//     Drive/Outputs/Out/nCtrl1 @bit 2 <-> STM Control/Control/Reduce torque
//     Drive/Outputs/Out/nCtrl1 @bit 1 <-> STM Control/Control/Reset
//     Drive/Outputs/Out/nDataOut2[0] <-> STM Velocity/Velocity
//   (this object) <-> PLC Rail (EtherCAT)/Power (EK1200)/PLC Junction 2 (EK1122)/IM2L0 AT2L0 SL1L0 JUNCTION (CU1124)/X1 PF1L0-WFS (EK1100)/PF1L0-EL5042
//     Enc/Inputs/In/nComState @bit 1 <-> WcState/InputToggle
//     Enc/Inputs/In/nComState <-> WcState/WcState
//     Enc/Inputs/In/nDataIn1 <-> FB Inputs Channel 2/Position
//     Enc/Inputs/In/nState1 @bit 12 <-> FB Inputs Channel 2/Status/Diag
//     Enc/Inputs/In/nState1 @bit 1 <-> FB Inputs Channel 2/Status/Error
//     Enc/Inputs/In/nState1 @bit 14 <-> FB Inputs Channel 2/Status/Input cycle counter
//     Enc/Inputs/In/nState1 @bit 2 <-> FB Inputs Channel 2/Status/Ready
//     Enc/Inputs/In/nState1 @bit 13 <-> FB Inputs Channel 2/Status/TxPDO State
//     Enc/Inputs/In/nState1 <-> FB Inputs Channel 2/Status/Warning
//   (this object) <-> PLC Rail (EtherCAT)/Power (EK1200)/PLC Junction 2 (EK1122)/IM2L0 AT2L0 SL1L0 JUNCTION (CU1124)/X1 PF1L0-WFS (EK1100)/PF1L0-EL7041-01
//     Drive/Inputs/In/nState1 @bit 3 <-> STM Status/Status/Error
//     Drive/Inputs/In/nState1 @bit 5 <-> STM Status/Status/Moving negative
//     Drive/Inputs/In/nState1 @bit 4 <-> STM Status/Status/Moving positive
//     Drive/Inputs/In/nState1 @bit 1 <-> STM Status/Status/Ready
//     Drive/Inputs/In/nState1 <-> STM Status/Status/Ready to enable
//     Drive/Inputs/In/nState1 @bit 6 <-> STM Status/Status/Torque reduced
//     Drive/Inputs/In/nState1 @bit 2 <-> STM Status/Status/Warning
//     Drive/Inputs/In/nState2 @bit 3 <-> STM Status/Status/Digital input 1
//     Drive/Inputs/In/nState2 @bit 4 <-> STM Status/Status/Digital input 2
//     Drive/Inputs/In/nState2 @bit 5 <-> STM Status/Status/Sync error
//     Drive/Inputs/In/nState2 @bit 7 <-> STM Status/Status/TxPDO Toggle
//     Drive/Inputs/In/nState4 @bit 1 <-> WcState/InputToggle
//     Drive/Inputs/In/nState4 <-> WcState/WcState
//     Drive/Outputs/Out/nCtrl1 <-> STM Control/Control/Enable
//     Drive/Outputs/Out/nCtrl1 @bit 2 <-> STM Control/Control/Reduce torque
//     Drive/Outputs/Out/nCtrl1 @bit 1 <-> STM Control/Control/Reset
//     Drive/Outputs/Out/nDataOut2[0] <-> STM Velocity/Velocity
//   (this object) <-> PLC Rail (EtherCAT)/Power (EK1200)/PLC Junction 1 (EK1122)/X1 RTDSL0 (EK1100)/RTDSL0-EL7041-01
//     Drive/Inputs/In/nState1 @bit 3 <-> STM Status/Status/Error
//     Drive/Inputs/In/nState1 @bit 5 <-> STM Status/Status/Moving negative
//     Drive/Inputs/In/nState1 @bit 4 <-> STM Status/Status/Moving positive
//     Drive/Inputs/In/nState1 @bit 1 <-> STM Status/Status/Ready
//     Drive/Inputs/In/nState1 <-> STM Status/Status/Ready to enable
//     Drive/Inputs/In/nState1 @bit 6 <-> STM Status/Status/Torque reduced
//     Drive/Inputs/In/nState1 @bit 2 <-> STM Status/Status/Warning
//     Drive/Inputs/In/nState2 @bit 3 <-> STM Status/Status/Digital input 1
//     Drive/Inputs/In/nState2 @bit 4 <-> STM Status/Status/Digital input 2
//     Drive/Inputs/In/nState2 @bit 5 <-> STM Status/Status/Sync error
//     Drive/Inputs/In/nState2 @bit 7 <-> STM Status/Status/TxPDO Toggle
//     Drive/Inputs/In/nState4 @bit 1 <-> WcState/InputToggle
//     Drive/Inputs/In/nState4 <-> WcState/WcState
//     Drive/Outputs/Out/nCtrl1 <-> STM Control/Control/Enable
//     Drive/Outputs/Out/nCtrl1 @bit 2 <-> STM Control/Control/Reduce torque
//     Drive/Outputs/Out/nCtrl1 @bit 1 <-> STM Control/Control/Reset
//     Drive/Outputs/Out/nDataOut2[0] <-> STM Velocity/Velocity
//     Enc/Inputs/In/nDataIn1[0] <-> ENC Status compact/Counter value
//     Enc/Inputs/In/nDataIn2[0] <-> ENC Status compact/Latch value
//     Enc/Inputs/In/nState1 @bit 4 <-> ENC Status compact/Status/Counter overflow
//     Enc/Inputs/In/nState1 @bit 3 <-> ENC Status compact/Status/Counter underflow
//     Enc/Inputs/In/nState1 @bit 7 <-> ENC Status compact/Status/Extrapolation stall
//     Enc/Inputs/In/nState1 <-> ENC Status compact/Status/Latch C valid
//     Enc/Inputs/In/nState1 @bit 1 <-> ENC Status compact/Status/Latch extern valid
//     Enc/Inputs/In/nState1 @bit 2 <-> ENC Status compact/Status/Set counter done
//     Enc/Inputs/In/nState2 @bit 4 <-> ENC Status compact/Status/Status of extern latch
//     Enc/Inputs/In/nState2 <-> ENC Status compact/Status/Status of input A
//     Enc/Inputs/In/nState2 @bit 1 <-> ENC Status compact/Status/Status of input B
//     Enc/Inputs/In/nState2 @bit 2 <-> ENC Status compact/Status/Status of input C
//     Enc/Inputs/In/nState2 @bit 5 <-> ENC Status compact/Status/Sync error
//     Enc/Inputs/In/nState2 @bit 7 <-> ENC Status compact/Status/TxPDO Toggle
//     Enc/Inputs/In/nState4 @bit 1 <-> WcState/InputToggle
//     Enc/Inputs/In/nState4 <-> WcState/WcState
//     Enc/Outputs/Out/nCtrl1 <-> ENC Control compact/Control/Enable latch C
//     Enc/Outputs/Out/nCtrl1 @bit 3 <-> ENC Control compact/Control/Enable latch extern on negative edge
//     Enc/Outputs/Out/nCtrl1 @bit 1 <-> ENC Control compact/Control/Enable latch extern on positive edge
//     Enc/Outputs/Out/nCtrl1 @bit 2 <-> ENC Control compact/Control/Set counter
//     Enc/Outputs/Out/nDataOut1[0] <-> ENC Control compact/Set counter value
//   (this object) <-> PLC Rail (EtherCAT)/Power (EK1200)/PLC Junction 1 (EK1122)/X1 RTDSL0 (EK1100)/RTDSL0-EL7041-05
//     Drive/Inputs/In/nState1 @bit 3 <-> STM Status/Status/Error
//     Drive/Inputs/In/nState1 @bit 5 <-> STM Status/Status/Moving negative
//     Drive/Inputs/In/nState1 @bit 4 <-> STM Status/Status/Moving positive
//     Drive/Inputs/In/nState1 @bit 1 <-> STM Status/Status/Ready
//     Drive/Inputs/In/nState1 <-> STM Status/Status/Ready to enable
//     Drive/Inputs/In/nState1 @bit 6 <-> STM Status/Status/Torque reduced
//     Drive/Inputs/In/nState1 @bit 2 <-> STM Status/Status/Warning
//     Drive/Inputs/In/nState2 @bit 3 <-> STM Status/Status/Digital input 1
//     Drive/Inputs/In/nState2 @bit 4 <-> STM Status/Status/Digital input 2
//     Drive/Inputs/In/nState2 @bit 5 <-> STM Status/Status/Sync error
//     Drive/Inputs/In/nState2 @bit 7 <-> STM Status/Status/TxPDO Toggle
//     Drive/Inputs/In/nState4 @bit 1 <-> WcState/InputToggle
//     Drive/Inputs/In/nState4 <-> WcState/WcState
//     Drive/Outputs/Out/nCtrl1 <-> STM Control/Control/Enable
//     Drive/Outputs/Out/nCtrl1 @bit 2 <-> STM Control/Control/Reduce torque
//     Drive/Outputs/Out/nCtrl1 @bit 1 <-> STM Control/Control/Reset
//     Drive/Outputs/Out/nDataOut2[0] <-> STM Velocity/Velocity
//   (this object) <-> PLC Rail (EtherCAT)/Power (EK1200)/PLC Junction 1 (EK1122)/X1 RTDSL0 (EK1100)/Term 113 (EL3054)
//     Enc/Inputs/In/nDataIn1[0] <-> AI Standard Channel 1/Value
//     Enc/Inputs/In/nState4 @bit 1 <-> WcState/InputToggle
//     Enc/Inputs/In/nState4 <-> WcState/WcState
//   (this object) <-> PLC Rail (EtherCAT)/Power (EK1200)/PLC Junction 2 (EK1122)/IM2L0 AT2L0 SL1L0 JUNCTION (CU1124)/X1 SL1L0-Power (EK1100)/SL1L0-EL5042-E2
//     Enc/Inputs/In/nComState @bit 1 <-> WcState/InputToggle
//     Enc/Inputs/In/nComState <-> WcState/WcState
//     Enc/Inputs/In/nDataIn1 <-> FB Inputs Channel 1/Position
//     Enc/Inputs/In/nDataIn1 <-> FB Inputs Channel 2/Position
//     Enc/Inputs/In/nState1 @bit 12 <-> FB Inputs Channel 1/Status/Diag
//     Enc/Inputs/In/nState1 @bit 12 <-> FB Inputs Channel 2/Status/Diag
//     Enc/Inputs/In/nState1 @bit 1 <-> FB Inputs Channel 1/Status/Error
//     Enc/Inputs/In/nState1 @bit 1 <-> FB Inputs Channel 2/Status/Error
//     Enc/Inputs/In/nState1 @bit 14 <-> FB Inputs Channel 1/Status/Input cycle counter
//     Enc/Inputs/In/nState1 @bit 14 <-> FB Inputs Channel 2/Status/Input cycle counter
//     Enc/Inputs/In/nState1 @bit 2 <-> FB Inputs Channel 1/Status/Ready
//     Enc/Inputs/In/nState1 @bit 2 <-> FB Inputs Channel 2/Status/Ready
//     Enc/Inputs/In/nState1 @bit 13 <-> FB Inputs Channel 1/Status/TxPDO State
//     Enc/Inputs/In/nState1 @bit 13 <-> FB Inputs Channel 2/Status/TxPDO State
//     Enc/Inputs/In/nState1 <-> FB Inputs Channel 1/Status/Warning
//     Enc/Inputs/In/nState1 <-> FB Inputs Channel 2/Status/Warning
//   (this object) <-> PLC Rail (EtherCAT)/Power (EK1200)/PLC Junction 2 (EK1122)/IM2L0 AT2L0 SL1L0 JUNCTION (CU1124)/X1 SL1L0-Power (EK1100)/SL1L0-EL7041-E1
//     Drive/Inputs/In/nState1 @bit 3 <-> STM Status/Status/Error
//     Drive/Inputs/In/nState1 @bit 5 <-> STM Status/Status/Moving negative
//     Drive/Inputs/In/nState1 @bit 4 <-> STM Status/Status/Moving positive
//     Drive/Inputs/In/nState1 @bit 1 <-> STM Status/Status/Ready
//     Drive/Inputs/In/nState1 <-> STM Status/Status/Ready to enable
//     Drive/Inputs/In/nState1 @bit 6 <-> STM Status/Status/Torque reduced
//     Drive/Inputs/In/nState1 @bit 2 <-> STM Status/Status/Warning
//     Drive/Inputs/In/nState2 @bit 3 <-> STM Status/Status/Digital input 1
//     Drive/Inputs/In/nState2 @bit 4 <-> STM Status/Status/Digital input 2
//     Drive/Inputs/In/nState2 @bit 5 <-> STM Status/Status/Sync error
//     Drive/Inputs/In/nState2 @bit 7 <-> STM Status/Status/TxPDO Toggle
//     Drive/Inputs/In/nState4 @bit 1 <-> WcState/InputToggle
//     Drive/Inputs/In/nState4 <-> WcState/WcState
//     Drive/Outputs/Out/nCtrl1 <-> STM Control/Control/Enable
//     Drive/Outputs/Out/nCtrl1 @bit 2 <-> STM Control/Control/Reduce torque
//     Drive/Outputs/Out/nCtrl1 @bit 1 <-> STM Control/Control/Reset
//     Drive/Outputs/Out/nDataOut2[0] <-> STM Velocity/Velocity
//   (this object) <-> PLC Rail (EtherCAT)/Power (EK1200)/PLC Junction 2 (EK1122)/IM2L0 AT2L0 SL1L0 JUNCTION (CU1124)/X1 SL1L0-Power (EK1100)/SL1L0-EL7041-E3
//     Drive/Inputs/In/nState1 @bit 3 <-> STM Status/Status/Error
//     Drive/Inputs/In/nState1 @bit 5 <-> STM Status/Status/Moving negative
//     Drive/Inputs/In/nState1 @bit 4 <-> STM Status/Status/Moving positive
//     Drive/Inputs/In/nState1 @bit 1 <-> STM Status/Status/Ready
//     Drive/Inputs/In/nState1 <-> STM Status/Status/Ready to enable
//     Drive/Inputs/In/nState1 @bit 6 <-> STM Status/Status/Torque reduced
//     Drive/Inputs/In/nState1 @bit 2 <-> STM Status/Status/Warning
//     Drive/Inputs/In/nState2 @bit 3 <-> STM Status/Status/Digital input 1
//     Drive/Inputs/In/nState2 @bit 4 <-> STM Status/Status/Digital input 2
//     Drive/Inputs/In/nState2 @bit 5 <-> STM Status/Status/Sync error
//     Drive/Inputs/In/nState2 @bit 7 <-> STM Status/Status/TxPDO Toggle
//     Drive/Inputs/In/nState4 @bit 1 <-> WcState/InputToggle
//     Drive/Inputs/In/nState4 <-> WcState/WcState
//     Drive/Outputs/Out/nCtrl1 <-> STM Control/Control/Enable
//     Drive/Outputs/Out/nCtrl1 @bit 2 <-> STM Control/Control/Reduce torque
//     Drive/Outputs/Out/nCtrl1 @bit 1 <-> STM Control/Control/Reset
//     Drive/Outputs/Out/nDataOut2[0] <-> STM Velocity/Velocity
//   (this object) <-> PLC Rail (EtherCAT)/Power (EK1200)/PLC Junction 2 (EK1122)/IM2L0 AT2L0 SL1L0 JUNCTION (CU1124)/X1 SL1L0-Power (EK1100)/SL1L0-EL5042-E6
//     Enc/Inputs/In/nComState @bit 1 <-> WcState/InputToggle
//     Enc/Inputs/In/nComState <-> WcState/WcState
//     Enc/Inputs/In/nDataIn1 <-> FB Inputs Channel 1/Position
//     Enc/Inputs/In/nDataIn1 <-> FB Inputs Channel 2/Position
//     Enc/Inputs/In/nState1 @bit 12 <-> FB Inputs Channel 1/Status/Diag
//     Enc/Inputs/In/nState1 @bit 12 <-> FB Inputs Channel 2/Status/Diag
//     Enc/Inputs/In/nState1 @bit 1 <-> FB Inputs Channel 1/Status/Error
//     Enc/Inputs/In/nState1 @bit 1 <-> FB Inputs Channel 2/Status/Error
//     Enc/Inputs/In/nState1 @bit 14 <-> FB Inputs Channel 1/Status/Input cycle counter
//     Enc/Inputs/In/nState1 @bit 14 <-> FB Inputs Channel 2/Status/Input cycle counter
//     Enc/Inputs/In/nState1 @bit 2 <-> FB Inputs Channel 1/Status/Ready
//     Enc/Inputs/In/nState1 @bit 2 <-> FB Inputs Channel 2/Status/Ready
//     Enc/Inputs/In/nState1 @bit 13 <-> FB Inputs Channel 1/Status/TxPDO State
//     Enc/Inputs/In/nState1 @bit 13 <-> FB Inputs Channel 2/Status/TxPDO State
//     Enc/Inputs/In/nState1 <-> FB Inputs Channel 1/Status/Warning
//     Enc/Inputs/In/nState1 <-> FB Inputs Channel 2/Status/Warning
//   (this object) <-> PLC Rail (EtherCAT)/Power (EK1200)/PLC Junction 2 (EK1122)/IM2L0 AT2L0 SL1L0 JUNCTION (CU1124)/X1 SL1L0-Power (EK1100)/SL1L0-EL7041-E5
//     Drive/Inputs/In/nState1 @bit 3 <-> STM Status/Status/Error
//     Drive/Inputs/In/nState1 @bit 5 <-> STM Status/Status/Moving negative
//     Drive/Inputs/In/nState1 @bit 4 <-> STM Status/Status/Moving positive
//     Drive/Inputs/In/nState1 @bit 1 <-> STM Status/Status/Ready
//     Drive/Inputs/In/nState1 <-> STM Status/Status/Ready to enable
//     Drive/Inputs/In/nState1 @bit 6 <-> STM Status/Status/Torque reduced
//     Drive/Inputs/In/nState1 @bit 2 <-> STM Status/Status/Warning
//     Drive/Inputs/In/nState2 @bit 3 <-> STM Status/Status/Digital input 1
//     Drive/Inputs/In/nState2 @bit 4 <-> STM Status/Status/Digital input 2
//     Drive/Inputs/In/nState2 @bit 5 <-> STM Status/Status/Sync error
//     Drive/Inputs/In/nState2 @bit 7 <-> STM Status/Status/TxPDO Toggle
//     Drive/Inputs/In/nState4 @bit 1 <-> WcState/InputToggle
//     Drive/Inputs/In/nState4 <-> WcState/WcState
//     Drive/Outputs/Out/nCtrl1 <-> STM Control/Control/Enable
//     Drive/Outputs/Out/nCtrl1 @bit 2 <-> STM Control/Control/Reduce torque
//     Drive/Outputs/Out/nCtrl1 @bit 1 <-> STM Control/Control/Reset
//     Drive/Outputs/Out/nDataOut2[0] <-> STM Velocity/Velocity
//   (this object) <-> PLC Rail (EtherCAT)/Power (EK1200)/PLC Junction 2 (EK1122)/IM2L0 AT2L0 SL1L0 JUNCTION (CU1124)/X1 SL1L0-Power (EK1100)/SL1L0-EL7041-E7
//     Drive/Inputs/In/nState1 @bit 3 <-> STM Status/Status/Error
//     Drive/Inputs/In/nState1 @bit 5 <-> STM Status/Status/Moving negative
//     Drive/Inputs/In/nState1 @bit 4 <-> STM Status/Status/Moving positive
//     Drive/Inputs/In/nState1 @bit 1 <-> STM Status/Status/Ready
//     Drive/Inputs/In/nState1 <-> STM Status/Status/Ready to enable
//     Drive/Inputs/In/nState1 @bit 6 <-> STM Status/Status/Torque reduced
//     Drive/Inputs/In/nState1 @bit 2 <-> STM Status/Status/Warning
//     Drive/Inputs/In/nState2 @bit 3 <-> STM Status/Status/Digital input 1
//     Drive/Inputs/In/nState2 @bit 4 <-> STM Status/Status/Digital input 2
//     Drive/Inputs/In/nState2 @bit 5 <-> STM Status/Status/Sync error
//     Drive/Inputs/In/nState2 @bit 7 <-> STM Status/Status/TxPDO Toggle
//     Drive/Inputs/In/nState4 @bit 1 <-> WcState/InputToggle
//     Drive/Inputs/In/nState4 <-> WcState/WcState
//     Drive/Outputs/Out/nCtrl1 <-> STM Control/Control/Enable
//     Drive/Outputs/Out/nCtrl1 @bit 2 <-> STM Control/Control/Reduce torque
//     Drive/Outputs/Out/nCtrl1 @bit 1 <-> STM Control/Control/Reset
//     Drive/Outputs/Out/nDataOut2[0] <-> STM Velocity/Velocity
//   lfe_motion Instance <-> PLC Rail (EtherCAT)/Power (EK1200)/PLC Junction 1 (EK1122)/X1 RTDSL0 (EK1100)/RTDSL0-EL7041-01
//     PlcTask Inputs/Main.M33.bLimitBackwardEnable <-> STM Status/Status/Digital input 2
//     PlcTask Inputs/Main.M33.bLimitForwardEnable <-> STM Status/Status/Digital input 1
//   lfe_motion Instance <-> PLC Rail (EtherCAT)/Power (EK1200)/PLC Junction 1 (EK1122)/X1 RTDSL0 (EK1100)/RTDSL0-EL7041-05
//     PlcTask Inputs/Main.M38.bLimitBackwardEnable <-> STM Status/Status/Digital input 2
//     PlcTask Inputs/Main.M38.bLimitForwardEnable <-> STM Status/Status/Digital input 1
//   lfe_motion Instance <-> PLC Rail (EtherCAT)/Power (EK1200)/PLC Junction 1 (EK1122)/X1 RTDSL0 (EK1100)/RTDSL0-MPA-EL1008
//     PlcTask Inputs/RTDSL0.RTDSL0_MPA_01.i_xInsertedLS <-> Channel 1/Input
//     PlcTask Inputs/RTDSL0.RTDSL0_MPA_02.i_xInsertedLS <-> Channel 3/Input
//     PlcTask Inputs/RTDSL0.RTDSL0_MPA_03.i_xInsertedLS <-> Channel 5/Input
//     PlcTask Inputs/RTDSL0.RTDSL0_MPA_04.i_xInsertedLS <-> Channel 7/Input
//     PlcTask Inputs/RTDSL0.RTDSL0_MPA_01.i_xRetractedLS <-> Channel 2/Input
//     PlcTask Inputs/RTDSL0.RTDSL0_MPA_02.i_xRetractedLS <-> Channel 4/Input
//     PlcTask Inputs/RTDSL0.RTDSL0_MPA_03.i_xRetractedLS <-> Channel 6/Input
//     PlcTask Inputs/RTDSL0.RTDSL0_MPA_04.i_xRetractedLS <-> Channel 8/Input
//   lfe_motion Instance <-> PLC Rail (EtherCAT)/Power (EK1200)/PLC Junction 1 (EK1122)/X1 RTDSL0 (EK1100)/RTDSL0-MPA-EL2008
//     PlcTask Outputs/RTDSL0.RTDSL0_MPA_01.q_xInsert_DO <-> Channel 1/Output
//     PlcTask Outputs/RTDSL0.RTDSL0_MPA_02.q_xInsert_DO <-> Channel 3/Output
//     PlcTask Outputs/RTDSL0.RTDSL0_MPA_03.q_xInsert_DO <-> Channel 5/Output
//     PlcTask Outputs/RTDSL0.RTDSL0_MPA_04.q_xInsert_DO <-> Channel 7/Output
//     PlcTask Outputs/RTDSL0.RTDSL0_MPA_01.q_xRetract_DO <-> Channel 2/Output
//     PlcTask Outputs/RTDSL0.RTDSL0_MPA_02.q_xRetract_DO <-> Channel 4/Output
//     PlcTask Outputs/RTDSL0.RTDSL0_MPA_03.q_xRetract_DO <-> Channel 6/Output
//     PlcTask Outputs/RTDSL0.RTDSL0_MPA_04.q_xRetract_DO <-> Channel 8/Output
//   lfe_motion Instance <-> PLC Rail (EtherCAT)/Power (EK1200)/PLC Junction 1 (EK1122)/X1 RTDSL0 (EK1100)/Term 113 (EL3054)
//     PlcTask Inputs/Main.M38.nRawEncoderINT <-> AI Standard Channel 1/Value
//   lfe_motion Instance <-> PLC Rail (EtherCAT)/Power (EK1200)/PLC Junction 1 (EK1122)/X2 IM1L0-XTES (EK1100)/IM1L0-EL1088
//     PlcTask Inputs/Main.M21.bHome <-> Channel 2/Input
//     PlcTask Inputs/Main.M22.bHome <-> Channel 4/Input
//     PlcTask Inputs/PRG_IM1L0_XTES.fbIM1L0.bFocusEndBwd <-> Channel 4/Input
//     PlcTask Inputs/PRG_IM1L0_XTES.fbIM1L0.bFocusEndFwd <-> Channel 3/Input
//     PlcTask Inputs/PRG_IM1L0_XTES.fbIM1L0.bZoomEndBwd <-> Channel 2/Input
//     PlcTask Inputs/PRG_IM1L0_XTES.fbIM1L0.bZoomEndFwd <-> Channel 1/Input
//   lfe_motion Instance <-> PLC Rail (EtherCAT)/Power (EK1200)/PLC Junction 1 (EK1122)/X2 IM1L0-XTES (EK1100)/IM1L0-EL2004
//     PlcTask Outputs/Main.M20.bBrakeRelease <-> Channel 1/Output
//     PlcTask Outputs/PRG_IM1L0_XTES.fbIM1L0.fbLED.bLEDPower <-> Channel 3/Output
//     PlcTask Outputs/PRG_IM1L0_XTES.fbIM1L0.fbOpal.bOpalPower <-> Channel 2/Output
//   lfe_motion Instance <-> PLC Rail (EtherCAT)/Power (EK1200)/PLC Junction 1 (EK1122)/X2 IM1L0-XTES (EK1100)/IM1L0-EL6002
//     PlcTask Inputs/PRG_IM1L0_XTES.stEL6In/D[{0..21}] <-> COM TxPDO-Map Inputs Channel 1/Data In {0..21}  (22 links)
//     PlcTask Inputs/PRG_IM1L0_XTES.stEL6In/Status <-> COM TxPDO-Map Inputs Channel 1/Status
//     PlcTask Outputs/PRG_IM1L0_XTES.stEL6Out/Ctrl <-> COM RxPDO-Map Outputs Channel 1/Ctrl
//     PlcTask Outputs/PRG_IM1L0_XTES.stEL6Out/D[{0..21}] <-> COM RxPDO-Map Outputs Channel 1/Data Out {0..21}  (22 links)
//   lfe_motion Instance <-> PLC Rail (EtherCAT)/Power (EK1200)/PLC Junction 1 (EK1122)/X2 IM1L0-XTES (EK1100)/IM1L0-EL7041
//     PlcTask Inputs/Main.M20.bLimitForwardEnable <-> STM Status/Status/Digital input 1
//   lfe_motion Instance <-> PLC Rail (EtherCAT)/Power (EK1200)/PLC Junction 1 (EK1122)/X2 IM1L0-XTES (EK1100)/IM1L0-EL7342
//     PlcTask Inputs/PRG_IM1L0_XTES.bIM1L0FlowOk <-> DCM Status Channel 1/Status/Digital input 1
//   lfe_motion Instance <-> PLC Rail (EtherCAT)/Power (EK1200)/PLC Junction 2 (EK1122)/IM2L0 AT2L0 SL1L0 JUNCTION (CU1124)/X1 IM2L0-XTES (EK1100)/IM2L0-EL1088
//     PlcTask Inputs/Main.M25.bHome <-> Channel 2/Input
//     PlcTask Inputs/Main.M26.bHome <-> Channel 4/Input
//     PlcTask Inputs/PRG_IM2L0_XTES.fbIM2L0.bFocusEndBwd <-> Channel 4/Input
//     PlcTask Inputs/PRG_IM2L0_XTES.fbIM2L0.bFocusEndFwd <-> Channel 3/Input
//     PlcTask Inputs/PRG_IM2L0_XTES.fbIM2L0.bZoomEndBwd <-> Channel 2/Input
//     PlcTask Inputs/PRG_IM2L0_XTES.fbIM2L0.bZoomEndFwd <-> Channel 1/Input
//   lfe_motion Instance <-> PLC Rail (EtherCAT)/Power (EK1200)/PLC Junction 2 (EK1122)/IM2L0 AT2L0 SL1L0 JUNCTION (CU1124)/X1 IM2L0-XTES (EK1100)/IM2L0-EL2004
//     PlcTask Outputs/Main.M24.bBrakeRelease <-> Channel 1/Output
//     PlcTask Outputs/PRG_IM2L0_XTES.fbIM2L0.fbLED.bLEDPower <-> Channel 3/Output
//     PlcTask Outputs/PRG_IM2L0_XTES.fbIM2L0.fbOpal.bOpalPower <-> Channel 2/Output
//   lfe_motion Instance <-> PLC Rail (EtherCAT)/Power (EK1200)/PLC Junction 2 (EK1122)/IM2L0 AT2L0 SL1L0 JUNCTION (CU1124)/X1 IM2L0-XTES (EK1100)/IM2L0-EL6002
//     PlcTask Inputs/PRG_IM2L0_XTES.stEL6In/D[{0..21}] <-> COM TxPDO-Map Inputs Channel 1/Data In {0..21}  (22 links)
//     PlcTask Inputs/PRG_IM2L0_XTES.stEL6In/Status <-> COM TxPDO-Map Inputs Channel 1/Status
//     PlcTask Outputs/PRG_IM2L0_XTES.stEL6Out/Ctrl <-> COM RxPDO-Map Outputs Channel 1/Ctrl
//     PlcTask Outputs/PRG_IM2L0_XTES.stEL6Out/D[{0..21}] <-> COM RxPDO-Map Outputs Channel 1/Data Out {0..21}  (22 links)
//   lfe_motion Instance <-> PLC Rail (EtherCAT)/Power (EK1200)/PLC Junction 2 (EK1122)/IM2L0 AT2L0 SL1L0 JUNCTION (CU1124)/X1 IM2L0-XTES (EK1100)/IM2L0-EL7041
//     PlcTask Inputs/PRG_IM2L0_XTES.bDefectiveLimitSwitch <-> STM Status/Status/Digital input 1
//   lfe_motion Instance <-> PLC Rail (EtherCAT)/Power (EK1200)/PLC Junction 2 (EK1122)/IM2L0 AT2L0 SL1L0 JUNCTION (CU1124)/X1 PF1L0-WFS (EK1100)/PF1L0-EL2004
//     PlcTask Outputs/Main.M31.bBrakeRelease <-> Channel 1/Output
//   lfe_motion Instance <-> PLC Rail (EtherCAT)/Power (EK1200)/PLC Junction 2 (EK1122)/IM2L0 AT2L0 SL1L0 JUNCTION (CU1124)/X1 PF1L0-WFS (EK1100)/PF1L0-EL3314
//     PlcTask Inputs/PRG_PF1L0_WFS.fbPF1L0.fbThermoCouple1.bError <-> TC Inputs Channel 1/Status/Error
//     PlcTask Inputs/PRG_PF1L0_WFS.fbPF1L0.fbThermoCouple2.bError <-> TC Inputs Channel 2/Status/Error
//     PlcTask Inputs/PRG_PF1L0_WFS.fbPF1L0.fbThermoCouple1.bOverrange <-> TC Inputs Channel 1/Status/Overrange
//     PlcTask Inputs/PRG_PF1L0_WFS.fbPF1L0.fbThermoCouple2.bOverrange <-> TC Inputs Channel 2/Status/Overrange
//     PlcTask Inputs/PRG_PF1L0_WFS.fbPF1L0.fbThermoCouple1.bUnderrange <-> TC Inputs Channel 1/Status/Underrange
//     PlcTask Inputs/PRG_PF1L0_WFS.fbPF1L0.fbThermoCouple2.bUnderrange <-> TC Inputs Channel 2/Status/Underrange
//     PlcTask Inputs/PRG_PF1L0_WFS.fbPF1L0.fbThermoCouple1.iRaw <-> TC Inputs Channel 1/Value
//     PlcTask Inputs/PRG_PF1L0_WFS.fbPF1L0.fbThermoCouple2.iRaw <-> TC Inputs Channel 2/Value
//   lfe_motion Instance <-> PLC Rail (EtherCAT)/Power (EK1200)/PLC Junction 2 (EK1122)/IM2L0 AT2L0 SL1L0 JUNCTION (CU1124)/X1 PF1L0-WFS (EK1100)/PF1L0-EL5042
//     PlcTask Inputs/Main.M31.nRawEncoderULINT <-> FB Inputs Channel 2/Position
//     PlcTask Inputs/Main.M32.nRawEncoderULINT <-> FB Inputs Channel 1/Position
//   lfe_motion Instance <-> PLC Rail (EtherCAT)/Power (EK1200)/PLC Junction 2 (EK1122)/IM2L0 AT2L0 SL1L0 JUNCTION (CU1124)/X1 PF1L0-WFS (EK1100)/PF1L0-EL7041-01
//     PlcTask Inputs/Main.M31.bLimitBackwardEnable <-> STM Status/Status/Digital input 2
//     PlcTask Inputs/Main.M31.bLimitForwardEnable <-> STM Status/Status/Digital input 1
//   lfe_motion Instance <-> PLC Rail (EtherCAT)/Power (EK1200)/PLC Junction 2 (EK1122)/IM2L0 AT2L0 SL1L0 JUNCTION (CU1124)/X1 SL1L0-Power (EK1100)/SL1L0-EL3202-E10
//     PlcTask Inputs/PRG_SL1L0_POWER.fbSL1L0.RTD_TOP_1.bError <-> RTD Inputs Channel 1/Status/Error
//     PlcTask Inputs/PRG_SL1L0_POWER.fbSL1L0.RTD_TOP_2.bError <-> RTD Inputs Channel 2/Status/Error
//     PlcTask Inputs/PRG_SL1L0_POWER.fbSL1L0.RTD_TOP_1.bOverrange <-> RTD Inputs Channel 1/Status/Overrange
//     PlcTask Inputs/PRG_SL1L0_POWER.fbSL1L0.RTD_TOP_2.bOverrange <-> RTD Inputs Channel 2/Status/Overrange
//     PlcTask Inputs/PRG_SL1L0_POWER.fbSL1L0.RTD_TOP_1.bUnderrange <-> RTD Inputs Channel 1/Status/Underrange
//     PlcTask Inputs/PRG_SL1L0_POWER.fbSL1L0.RTD_TOP_2.bUnderrange <-> RTD Inputs Channel 2/Status/Underrange
//     PlcTask Inputs/PRG_SL1L0_POWER.fbSL1L0.RTD_TOP_1.iRaw <-> RTD Inputs Channel 1/Value
//     PlcTask Inputs/PRG_SL1L0_POWER.fbSL1L0.RTD_TOP_2.iRaw <-> RTD Inputs Channel 2/Value
//   lfe_motion Instance <-> PLC Rail (EtherCAT)/Power (EK1200)/PLC Junction 2 (EK1122)/IM2L0 AT2L0 SL1L0 JUNCTION (CU1124)/X1 SL1L0-Power (EK1100)/SL1L0-EL3202-E11
//     PlcTask Inputs/PRG_SL1L0_POWER.fbSL1L0.RTD_North_1.bError <-> RTD Inputs Channel 1/Status/Error
//     PlcTask Inputs/PRG_SL1L0_POWER.fbSL1L0.RTD_North_2.bError <-> RTD Inputs Channel 2/Status/Error
//     PlcTask Inputs/PRG_SL1L0_POWER.fbSL1L0.RTD_North_1.bOverrange <-> RTD Inputs Channel 1/Status/Overrange
//     PlcTask Inputs/PRG_SL1L0_POWER.fbSL1L0.RTD_North_2.bOverrange <-> RTD Inputs Channel 2/Status/Overrange
//     PlcTask Inputs/PRG_SL1L0_POWER.fbSL1L0.RTD_North_1.bUnderrange <-> RTD Inputs Channel 1/Status/Underrange
//     PlcTask Inputs/PRG_SL1L0_POWER.fbSL1L0.RTD_North_2.bUnderrange <-> RTD Inputs Channel 2/Status/Underrange
//     PlcTask Inputs/PRG_SL1L0_POWER.fbSL1L0.RTD_North_1.iRaw <-> RTD Inputs Channel 1/Value
//     PlcTask Inputs/PRG_SL1L0_POWER.fbSL1L0.RTD_North_2.iRaw <-> RTD Inputs Channel 2/Value
//   lfe_motion Instance <-> PLC Rail (EtherCAT)/Power (EK1200)/PLC Junction 2 (EK1122)/IM2L0 AT2L0 SL1L0 JUNCTION (CU1124)/X1 SL1L0-Power (EK1100)/SL1L0-EL3202-E8
//     PlcTask Inputs/PRG_SL1L0_POWER.fbSL1L0.RTD_Bottom_1.bError <-> RTD Inputs Channel 1/Status/Error
//     PlcTask Inputs/PRG_SL1L0_POWER.fbSL1L0.RTD_Bottom_2.bError <-> RTD Inputs Channel 2/Status/Error
//     PlcTask Inputs/PRG_SL1L0_POWER.fbSL1L0.RTD_Bottom_1.bOverrange <-> RTD Inputs Channel 1/Status/Overrange
//     PlcTask Inputs/PRG_SL1L0_POWER.fbSL1L0.RTD_Bottom_2.bOverrange <-> RTD Inputs Channel 2/Status/Overrange
//     PlcTask Inputs/PRG_SL1L0_POWER.fbSL1L0.RTD_Bottom_1.bUnderrange <-> RTD Inputs Channel 1/Status/Underrange
//     PlcTask Inputs/PRG_SL1L0_POWER.fbSL1L0.RTD_Bottom_2.bUnderrange <-> RTD Inputs Channel 2/Status/Underrange
//     PlcTask Inputs/PRG_SL1L0_POWER.fbSL1L0.RTD_Bottom_1.iRaw <-> RTD Inputs Channel 1/Value
//     PlcTask Inputs/PRG_SL1L0_POWER.fbSL1L0.RTD_Bottom_2.iRaw <-> RTD Inputs Channel 2/Value
//   lfe_motion Instance <-> PLC Rail (EtherCAT)/Power (EK1200)/PLC Junction 2 (EK1122)/IM2L0 AT2L0 SL1L0 JUNCTION (CU1124)/X1 SL1L0-Power (EK1100)/SL1L0-EL3202-E9
//     PlcTask Inputs/PRG_SL1L0_POWER.fbSL1L0.RTD_South_1.bError <-> RTD Inputs Channel 1/Status/Error
//     PlcTask Inputs/PRG_SL1L0_POWER.fbSL1L0.RTD_South_2.bError <-> RTD Inputs Channel 2/Status/Error
//     PlcTask Inputs/PRG_SL1L0_POWER.fbSL1L0.RTD_South_1.bOverrange <-> RTD Inputs Channel 1/Status/Overrange
//     PlcTask Inputs/PRG_SL1L0_POWER.fbSL1L0.RTD_South_2.bOverrange <-> RTD Inputs Channel 2/Status/Overrange
//     PlcTask Inputs/PRG_SL1L0_POWER.fbSL1L0.RTD_South_1.bUnderrange <-> RTD Inputs Channel 1/Status/Underrange
//     PlcTask Inputs/PRG_SL1L0_POWER.fbSL1L0.RTD_South_2.bUnderrange <-> RTD Inputs Channel 2/Status/Underrange
//     PlcTask Inputs/PRG_SL1L0_POWER.fbSL1L0.RTD_South_1.iRaw <-> RTD Inputs Channel 1/Value
//     PlcTask Inputs/PRG_SL1L0_POWER.fbSL1L0.RTD_South_2.iRaw <-> RTD Inputs Channel 2/Value
//   lfe_motion Instance <-> PLC Rail (EtherCAT)/Power (EK1200)/PLC Junction 2 (EK1122)/IM2L0 AT2L0 SL1L0 JUNCTION (CU1124)/X1 SL1L0-Power (EK1100)/SL1L0-EL7041-E1
//     PlcTask Inputs/Main.M41.bLimitBackwardEnable <-> STM Status/Status/Digital input 1
//     PlcTask Inputs/Main.M41.bLimitForwardEnable <-> STM Status/Status/Digital input 2
//   lfe_motion Instance <-> PLC Rail (EtherCAT)/Power (EK1200)/PLC Junction 2 (EK1122)/IM2L0 AT2L0 SL1L0 JUNCTION (CU1124)/X1 SL1L0-Power (EK1100)/SL1L0-EL7041-E3
//     PlcTask Inputs/Main.M42.bLimitBackwardEnable <-> STM Status/Status/Digital input 2
//     PlcTask Inputs/Main.M42.bLimitForwardEnable <-> STM Status/Status/Digital input 1
//   lfe_motion Instance <-> PLC Rail (EtherCAT)/Power (EK1200)/PLC Junction 2 (EK1122)/IM2L0 AT2L0 SL1L0 JUNCTION (CU1124)/X1 SL1L0-Power (EK1100)/SL1L0-EL7041-E5
//     PlcTask Inputs/Main.M43.bLimitBackwardEnable <-> STM Status/Status/Digital input 1
//     PlcTask Inputs/Main.M43.bLimitForwardEnable <-> STM Status/Status/Digital input 2
//   lfe_motion Instance <-> PLC Rail (EtherCAT)/Power (EK1200)/PLC Junction 2 (EK1122)/IM2L0 AT2L0 SL1L0 JUNCTION (CU1124)/X1 SL1L0-Power (EK1100)/SL1L0-EL7041-E7
//     PlcTask Inputs/Main.M44.bLimitBackwardEnable <-> STM Status/Status/Digital input 2
//     PlcTask Inputs/Main.M44.bLimitForwardEnable <-> STM Status/Status/Digital input 1
//   lfe_motion Instance <-> PLC Rail (EtherCAT)/Power (EK1200)/PLC Junction 2 (EK1122)/IM2L0 AT2L0 SL1L0 JUNCTION (CU1124)/X2 AT2L0-SOLID (EK1100)/AT2L0-EL7041-01
//     PlcTask Inputs/Main.M1.bLimitBackwardEnable <-> STM Status/Status/Digital input 1
//     PlcTask Inputs/Main.M1.bLimitForwardEnable <-> STM Status/Status/Digital input 2
//   lfe_motion Instance <-> PLC Rail (EtherCAT)/Power (EK1200)/PLC Junction 2 (EK1122)/IM2L0 AT2L0 SL1L0 JUNCTION (CU1124)/X2 AT2L0-SOLID (EK1100)/AT2L0-EL7041-02
//     PlcTask Inputs/Main.M2.bLimitBackwardEnable <-> STM Status/Status/Digital input 1
//     PlcTask Inputs/Main.M2.bLimitForwardEnable <-> STM Status/Status/Digital input 2
//   lfe_motion Instance <-> PLC Rail (EtherCAT)/Power (EK1200)/PLC Junction 2 (EK1122)/IM2L0 AT2L0 SL1L0 JUNCTION (CU1124)/X2 AT2L0-SOLID (EK1100)/AT2L0-EL7041-03
//     PlcTask Inputs/Main.M3.bLimitBackwardEnable <-> STM Status/Status/Digital input 1
//     PlcTask Inputs/Main.M3.bLimitForwardEnable <-> STM Status/Status/Digital input 2
//   lfe_motion Instance <-> PLC Rail (EtherCAT)/Power (EK1200)/PLC Junction 2 (EK1122)/IM2L0 AT2L0 SL1L0 JUNCTION (CU1124)/X2 AT2L0-SOLID (EK1100)/AT2L0-EL7041-04
//     PlcTask Inputs/Main.M4.bLimitBackwardEnable <-> STM Status/Status/Digital input 1
//     PlcTask Inputs/Main.M4.bLimitForwardEnable <-> STM Status/Status/Digital input 2
//   lfe_motion Instance <-> PLC Rail (EtherCAT)/Power (EK1200)/PLC Junction 2 (EK1122)/IM2L0 AT2L0 SL1L0 JUNCTION (CU1124)/X2 AT2L0-SOLID (EK1100)/AT2L0-EL7041-05
//     PlcTask Inputs/Main.M5.bLimitBackwardEnable <-> STM Status/Status/Digital input 1
//     PlcTask Inputs/Main.M5.bLimitForwardEnable <-> STM Status/Status/Digital input 2
//   lfe_motion Instance <-> PLC Rail (EtherCAT)/Power (EK1200)/PLC Junction 2 (EK1122)/IM2L0 AT2L0 SL1L0 JUNCTION (CU1124)/X2 AT2L0-SOLID (EK1100)/AT2L0-EL7041-06
//     PlcTask Inputs/Main.M6.bLimitBackwardEnable <-> STM Status/Status/Digital input 1
//     PlcTask Inputs/Main.M6.bLimitForwardEnable <-> STM Status/Status/Digital input 2
//   lfe_motion Instance <-> PLC Rail (EtherCAT)/Power (EK1200)/PLC Junction 2 (EK1122)/IM2L0 AT2L0 SL1L0 JUNCTION (CU1124)/X2 AT2L0-SOLID (EK1100)/AT2L0-EL7041-07
//     PlcTask Inputs/Main.M7.bLimitBackwardEnable <-> STM Status/Status/Digital input 1
//     PlcTask Inputs/Main.M7.bLimitForwardEnable <-> STM Status/Status/Digital input 2
//   lfe_motion Instance <-> PLC Rail (EtherCAT)/Power (EK1200)/PLC Junction 2 (EK1122)/IM2L0 AT2L0 SL1L0 JUNCTION (CU1124)/X2 AT2L0-SOLID (EK1100)/AT2L0-EL7041-08
//     PlcTask Inputs/Main.M8.bLimitBackwardEnable <-> STM Status/Status/Digital input 1
//     PlcTask Inputs/Main.M8.bLimitForwardEnable <-> STM Status/Status/Digital input 2
//   lfe_motion Instance <-> PLC Rail (EtherCAT)/Power (EK1200)/PLC Junction 2 (EK1122)/IM2L0 AT2L0 SL1L0 JUNCTION (CU1124)/X2 AT2L0-SOLID (EK1100)/AT2L0-EL7041-09
//     PlcTask Inputs/Main.M9.bLimitBackwardEnable <-> STM Status/Status/Digital input 1
//     PlcTask Inputs/Main.M9.bLimitForwardEnable <-> STM Status/Status/Digital input 2
//   lfe_motion Instance <-> PLC Rail (EtherCAT)/Power (EK1200)/PLC Junction 2 (EK1122)/IM2L0 AT2L0 SL1L0 JUNCTION (CU1124)/X2 AT2L0-SOLID (EK1100)/AT2L0-EL7041-10
//     PlcTask Inputs/Main.M10.bLimitBackwardEnable <-> STM Status/Status/Digital input 1
//     PlcTask Inputs/Main.M10.bLimitForwardEnable <-> STM Status/Status/Digital input 2
//   lfe_motion Instance <-> PLC Rail (EtherCAT)/Power (EK1200)/PLC Junction 2 (EK1122)/IM2L0 AT2L0 SL1L0 JUNCTION (CU1124)/X2 AT2L0-SOLID (EK1100)/AT2L0-EL7041-11
//     PlcTask Inputs/Main.M11.bLimitBackwardEnable <-> STM Status/Status/Digital input 1
//     PlcTask Inputs/Main.M11.bLimitForwardEnable <-> STM Status/Status/Digital input 2
//   lfe_motion Instance <-> PLC Rail (EtherCAT)/Power (EK1200)/PLC Junction 2 (EK1122)/IM2L0 AT2L0 SL1L0 JUNCTION (CU1124)/X2 AT2L0-SOLID (EK1100)/AT2L0-EL7041-12
//     PlcTask Inputs/Main.M12.bLimitBackwardEnable <-> STM Status/Status/Digital input 1
//     PlcTask Inputs/Main.M12.bLimitForwardEnable <-> STM Status/Status/Digital input 2
//   lfe_motion Instance <-> PLC Rail (EtherCAT)/Power (EK1200)/PLC Junction 2 (EK1122)/IM2L0 AT2L0 SL1L0 JUNCTION (CU1124)/X2 AT2L0-SOLID (EK1100)/AT2L0-EL7041-13
//     PlcTask Inputs/Main.M13.bLimitBackwardEnable <-> STM Status/Status/Digital input 1
//     PlcTask Inputs/Main.M13.bLimitForwardEnable <-> STM Status/Status/Digital input 2
//   lfe_motion Instance <-> PLC Rail (EtherCAT)/Power (EK1200)/PLC Junction 2 (EK1122)/IM2L0 AT2L0 SL1L0 JUNCTION (CU1124)/X2 AT2L0-SOLID (EK1100)/AT2L0-EL7041-14
//     PlcTask Inputs/Main.M14.bLimitBackwardEnable <-> STM Status/Status/Digital input 1
//     PlcTask Inputs/Main.M14.bLimitForwardEnable <-> STM Status/Status/Digital input 2
//   lfe_motion Instance <-> PLC Rail (EtherCAT)/Power (EK1200)/PLC Junction 2 (EK1122)/IM2L0 AT2L0 SL1L0 JUNCTION (CU1124)/X2 AT2L0-SOLID (EK1100)/AT2L0-EL7041-15
//     PlcTask Inputs/Main.M15.bLimitBackwardEnable <-> STM Status/Status/Digital input 1
//     PlcTask Inputs/Main.M15.bLimitForwardEnable <-> STM Status/Status/Digital input 2
//   lfe_motion Instance <-> PLC Rail (EtherCAT)/Power (EK1200)/PLC Junction 2 (EK1122)/IM2L0 AT2L0 SL1L0 JUNCTION (CU1124)/X2 AT2L0-SOLID (EK1100)/AT2L0-EL7041-16
//     PlcTask Inputs/Main.M16.bLimitBackwardEnable <-> STM Status/Status/Digital input 1
//     PlcTask Inputs/Main.M16.bLimitForwardEnable <-> STM Status/Status/Digital input 2
//   lfe_motion Instance <-> PLC Rail (EtherCAT)/Power (EK1200)/PLC Junction 2 (EK1122)/IM2L0 AT2L0 SL1L0 JUNCTION (CU1124)/X2 AT2L0-SOLID (EK1100)/AT2L0-EL7041-17
//     PlcTask Inputs/Main.M17.bLimitBackwardEnable <-> STM Status/Status/Digital input 1
//     PlcTask Inputs/Main.M17.bLimitForwardEnable <-> STM Status/Status/Digital input 2
//   lfe_motion Instance <-> PLC Rail (EtherCAT)/Power (EK1200)/PLC Junction 2 (EK1122)/IM2L0 AT2L0 SL1L0 JUNCTION (CU1124)/X2 AT2L0-SOLID (EK1100)/AT2L0-EL7041-18
//     PlcTask Inputs/Main.M18.bLimitBackwardEnable <-> STM Status/Status/Digital input 1
//     PlcTask Inputs/Main.M18.bLimitForwardEnable <-> STM Status/Status/Digital input 2
//   lfe_motion Instance <-> PLC Rail (EtherCAT)/Power (EK1200)/PLC Junction 2 (EK1122)/IM2L0 AT2L0 SL1L0 JUNCTION (CU1124)/X2 AT2L0-SOLID (EK1100)/AT2L0-EL7041-19
//     PlcTask Inputs/Main.M19.bLimitBackwardEnable <-> STM Status/Status/Digital input 1
//     PlcTask Inputs/Main.M19.bLimitForwardEnable <-> STM Status/Status/Digital input 2
//   lfe_motion Instance <-> PLC Rail (EtherCAT)/Power (EK1200)/PLC Junction 2 (EK1122)/X2 HXR EC2 (EK1100)/EC2 E1 (EK1122)/X1 IM3L0-PPM (EK1100)/IM3L0-EL2004
//     PlcTask Outputs/Main.M27.bBrakeRelease <-> Channel 1/Output
//     PlcTask Outputs/PRG_IM3L0_PPM.fbIM3L0.fbGige.bGigePower <-> Channel 2/Output
//   lfe_motion Instance <-> PLC Rail (EtherCAT)/Power (EK1200)/PLC Junction 2 (EK1122)/X2 HXR EC2 (EK1100)/EC2 E1 (EK1122)/X1 IM3L0-PPM (EK1100)/IM3L0-EL3062
//     PlcTask Inputs/PRG_IM3L0_PPM.fbIM3L0.fbPowerMeter.iVoltageINT <-> AI Standard Channel 1/Value
//   lfe_motion Instance <-> PLC Rail (EtherCAT)/Power (EK1200)/PLC Junction 2 (EK1122)/X2 HXR EC2 (EK1100)/EC2 E1 (EK1122)/X1 IM3L0-PPM (EK1100)/IM3L0-EL3314
//     PlcTask Inputs/PRG_IM3L0_PPM.fbIM3L0.fbPowerMeter.fbTempSensor.bError <-> TC Inputs Channel 1/Status/Error
//     PlcTask Inputs/PRG_IM3L0_PPM.fbIM3L0.fbPowerMeter.fbTempSensor.bOverrange <-> TC Inputs Channel 1/Status/Overrange
//     PlcTask Inputs/PRG_IM3L0_PPM.fbIM3L0.fbPowerMeter.fbTempSensor.bUnderrange <-> TC Inputs Channel 1/Status/Underrange
//     PlcTask Inputs/PRG_IM3L0_PPM.fbIM3L0.fbPowerMeter.fbTempSensor.iRaw <-> TC Inputs Channel 1/Value
//     PlcTask Inputs/PRG_IM3L0_PPM.fbIM3L0.fbYagTempSensor.bError <-> TC Inputs Channel 2/Status/Error
//     PlcTask Inputs/PRG_IM3L0_PPM.fbIM3L0.fbYagTempSensor.bOverrange <-> TC Inputs Channel 2/Status/Overrange
//     PlcTask Inputs/PRG_IM3L0_PPM.fbIM3L0.fbYagTempSensor.bUnderrange <-> TC Inputs Channel 2/Status/Underrange
//     PlcTask Inputs/PRG_IM3L0_PPM.fbIM3L0.fbYagTempSensor.iRaw <-> TC Inputs Channel 2/Value
//   lfe_motion Instance <-> PLC Rail (EtherCAT)/Power (EK1200)/PLC Junction 2 (EK1122)/X2 HXR EC2 (EK1100)/EC2 E1 (EK1122)/X1 IM3L0-PPM (EK1100)/IM3L0-EL4004
//     PlcTask Outputs/PRG_IM3L0_PPM.fbIM3L0.fbGige.iIlluminatorINT <-> AO Outputs Channel 1/Analog output
//   lfe_motion Instance <-> PLC Rail (EtherCAT)/Power (EK1200)/PLC Junction 2 (EK1122)/X2 HXR EC2 (EK1100)/EC2 E1 (EK1122)/X1 IM3L0-PPM (EK1100)/IM3L0-EL7041
//     PlcTask Inputs/Main.M27.bLimitBackwardEnable <-> STM Status/Status/Digital input 2
//     PlcTask Inputs/Main.M27.bLimitForwardEnable <-> STM Status/Status/Digital input 1
//   lfe_motion Instance <-> PLC Rail (EtherCAT)/Power (EK1200)/PLC Junction 2 (EK1122)/X2 HXR EC2 (EK1100)/EC2 E1 (EK1122)/X2 IM1L1-PPM (EK1100)/IM1L1-EL2004
//     PlcTask Outputs/Main.M23.bBrakeRelease <-> Channel 1/Output
//     PlcTask Outputs/PRG_IM1L1_PPM.fbIM1L1.fbGige.bGigePower <-> Channel 2/Output
//   lfe_motion Instance <-> PLC Rail (EtherCAT)/Power (EK1200)/PLC Junction 2 (EK1122)/X2 HXR EC2 (EK1100)/EC2 E1 (EK1122)/X2 IM1L1-PPM (EK1100)/IM1L1-EL3062
//     PlcTask Inputs/PRG_IM1L1_PPM.fbIM1L1.fbPowerMeter.iVoltageINT <-> AI Standard Channel 1/Value
//   lfe_motion Instance <-> PLC Rail (EtherCAT)/Power (EK1200)/PLC Junction 2 (EK1122)/X2 HXR EC2 (EK1100)/EC2 E1 (EK1122)/X2 IM1L1-PPM (EK1100)/IM1L1-EL3314
//     PlcTask Inputs/PRG_IM1L1_PPM.fbIM1L1.fbPowerMeter.fbTempSensor.bError <-> TC Inputs Channel 1/Status/Error
//     PlcTask Inputs/PRG_IM1L1_PPM.fbIM1L1.fbPowerMeter.fbTempSensor.bOverrange <-> TC Inputs Channel 1/Status/Overrange
//     PlcTask Inputs/PRG_IM1L1_PPM.fbIM1L1.fbPowerMeter.fbTempSensor.bUnderrange <-> TC Inputs Channel 1/Status/Underrange
//     PlcTask Inputs/PRG_IM1L1_PPM.fbIM1L1.fbPowerMeter.fbTempSensor.iRaw <-> TC Inputs Channel 1/Value
//     PlcTask Inputs/PRG_IM1L1_PPM.fbIM1L1.fbYagTempSensor.bError <-> TC Inputs Channel 2/Status/Error
//     PlcTask Inputs/PRG_IM1L1_PPM.fbIM1L1.fbYagTempSensor.bOverrange <-> TC Inputs Channel 2/Status/Overrange
//     PlcTask Inputs/PRG_IM1L1_PPM.fbIM1L1.fbYagTempSensor.bUnderrange <-> TC Inputs Channel 2/Status/Underrange
//     PlcTask Inputs/PRG_IM1L1_PPM.fbIM1L1.fbYagTempSensor.iRaw <-> TC Inputs Channel 2/Value
//   lfe_motion Instance <-> PLC Rail (EtherCAT)/Power (EK1200)/PLC Junction 2 (EK1122)/X2 HXR EC2 (EK1100)/EC2 E1 (EK1122)/X2 IM1L1-PPM (EK1100)/IM1L1-EL4004
//     PlcTask Outputs/PRG_IM1L1_PPM.fbIM1L1.fbGige.iIlluminatorINT <-> AO Outputs Channel 1/Analog output
//   lfe_motion Instance <-> PLC Rail (EtherCAT)/Power (EK1200)/PLC Junction 2 (EK1122)/X2 HXR EC2 (EK1100)/EC2 E1 (EK1122)/X2 IM1L1-PPM (EK1100)/IM1L1-EL7041
//     PlcTask Inputs/Main.M23.bLimitBackwardEnable <-> STM Status/Status/Digital input 2
//     PlcTask Inputs/Main.M23.bLimitForwardEnable <-> STM Status/Status/Digital input 1
//   lfe_motion Instance <-> PLC Rail (EtherCAT)/Power (EK1200)/PLC Junction 2 (EK1122)/X2 HXR EC2 (EK1100)/EC2 E2 (EK1122)/X1 IM4L0-XTES (EK1100)/IM4L0-EL1088
//     PlcTask Inputs/Main.M29.bHome <-> Channel 2/Input
//     PlcTask Inputs/Main.M30.bHome <-> Channel 4/Input
//     PlcTask Inputs/PRG_IM4L0_XTES.fbIM4L0.bFocusEndBwd <-> Channel 4/Input
//     PlcTask Inputs/PRG_IM4L0_XTES.fbIM4L0.bFocusEndFwd <-> Channel 3/Input
//     PlcTask Inputs/PRG_IM4L0_XTES.fbIM4L0.bZoomEndBwd <-> Channel 2/Input
//     PlcTask Inputs/PRG_IM4L0_XTES.fbIM4L0.bZoomEndFwd <-> Channel 1/Input
//   lfe_motion Instance <-> PLC Rail (EtherCAT)/Power (EK1200)/PLC Junction 2 (EK1122)/X2 HXR EC2 (EK1100)/EC2 E2 (EK1122)/X1 IM4L0-XTES (EK1100)/IM4L0-EL2004
//     PlcTask Outputs/Main.M28.bBrakeRelease <-> Channel 1/Output
//     PlcTask Outputs/PRG_IM4L0_XTES.bIM4L0_SCRP_LED_01 <-> Channel 4/Output
//     PlcTask Outputs/PRG_IM4L0_XTES.fbIM4L0.fbLED.bLEDPower <-> Channel 3/Output
//     PlcTask Outputs/PRG_IM4L0_XTES.fbIM4L0.fbOpal.bOpalPower <-> Channel 2/Output
//   lfe_motion Instance <-> PLC Rail (EtherCAT)/Power (EK1200)/PLC Junction 2 (EK1122)/X2 HXR EC2 (EK1100)/EC2 E2 (EK1122)/X1 IM4L0-XTES (EK1100)/IM4L0-EL6002
//     PlcTask Inputs/PRG_IM4L0_XTES.stEL6In/D[{0..21}] <-> COM TxPDO-Map Inputs Channel 1/Data In {0..21}  (22 links)
//     PlcTask Inputs/PRG_IM4L0_XTES.stEL6In/Status <-> COM TxPDO-Map Inputs Channel 1/Status
//     PlcTask Outputs/PRG_IM4L0_XTES.stEL6Out/Ctrl <-> COM RxPDO-Map Outputs Channel 1/Ctrl
//     PlcTask Outputs/PRG_IM4L0_XTES.stEL6Out/D[{0..21}] <-> COM RxPDO-Map Outputs Channel 1/Data Out {0..21}  (22 links)
//   lfe_motion Instance <-> PLC Rail (EtherCAT)/Power (EK1200)/PLC Junction 2 (EK1122)/X2 HXR EC2 (EK1100)/EC2 E2 (EK1122)/X1 IM4L0-XTES (EK1100)/IM4L0-EL7041
//     PlcTask Inputs/Main.M28.bLimitForwardEnable <-> STM Status/Status/Digital input 1
//   lfe_motion Instance <-> PLC Rail (EtherCAT)/Power (EK1200)/PLC Junction 2 (EK1122)/X2 SL2L0-Power (EK1100)/SL2L0-EL3202-E10
//     PlcTask Inputs/PRG_SL2L0_POWER.fbSL2L0.RTD_North_1.bError <-> RTD Inputs Channel 1/Status/Error
//     PlcTask Inputs/PRG_SL2L0_POWER.fbSL2L0.RTD_North_1.iRaw <-> RTD Inputs Channel 1/Value
//     PlcTask Inputs/PRG_SL2L0_POWER.fbSL2L0.RTD_TOP_1.bError <-> RTD Inputs Channel 1/Status/Error
//     PlcTask Inputs/PRG_SL2L0_POWER.fbSL2L0.RTD_TOP_2.bError <-> RTD Inputs Channel 2/Status/Error
//     PlcTask Inputs/PRG_SL2L0_POWER.fbSL2L0.RTD_TOP_1.bOverrange <-> RTD Inputs Channel 1/Status/Overrange
//     PlcTask Inputs/PRG_SL2L0_POWER.fbSL2L0.RTD_TOP_2.bOverrange <-> RTD Inputs Channel 2/Status/Overrange
//     PlcTask Inputs/PRG_SL2L0_POWER.fbSL2L0.RTD_TOP_1.bUnderrange <-> RTD Inputs Channel 1/Status/Underrange
//     PlcTask Inputs/PRG_SL2L0_POWER.fbSL2L0.RTD_TOP_2.bUnderrange <-> RTD Inputs Channel 2/Status/Underrange
//     PlcTask Inputs/PRG_SL2L0_POWER.fbSL2L0.RTD_TOP_1.iRaw <-> RTD Inputs Channel 1/Value
//     PlcTask Inputs/PRG_SL2L0_POWER.fbSL2L0.RTD_TOP_2.iRaw <-> RTD Inputs Channel 2/Value
//   lfe_motion Instance <-> PLC Rail (EtherCAT)/Power (EK1200)/PLC Junction 2 (EK1122)/X2 SL2L0-Power (EK1100)/SL2L0-EL3202-E11
//     PlcTask Inputs/PRG_SL2L0_POWER.fbSL2L0.RTD_North_1.bOverrange <-> RTD Inputs Channel 1/Status/Overrange
//     PlcTask Inputs/PRG_SL2L0_POWER.fbSL2L0.RTD_North_2.bOverrange <-> RTD Inputs Channel 2/Status/Overrange
//     PlcTask Inputs/PRG_SL2L0_POWER.fbSL2L0.RTD_North_1.bUnderrange <-> RTD Inputs Channel 1/Status/Underrange
//     PlcTask Inputs/PRG_SL2L0_POWER.fbSL2L0.RTD_North_2.bUnderrange <-> RTD Inputs Channel 2/Status/Underrange
//     PlcTask Inputs/PRG_SL2L0_POWER.fbSL2L0.RTD_North_2.bError <-> RTD Inputs Channel 2/Status/Error
//     PlcTask Inputs/PRG_SL2L0_POWER.fbSL2L0.RTD_North_2.iRaw <-> RTD Inputs Channel 2/Value
//   lfe_motion Instance <-> PLC Rail (EtherCAT)/Power (EK1200)/PLC Junction 2 (EK1122)/X2 SL2L0-Power (EK1100)/SL2L0-EL3202-E8
//     PlcTask Inputs/PRG_SL2L0_POWER.fbSL2L0.RTD_Bottom_1.bError <-> RTD Inputs Channel 1/Status/Error
//     PlcTask Inputs/PRG_SL2L0_POWER.fbSL2L0.RTD_Bottom_2.bError <-> RTD Inputs Channel 2/Status/Error
//     PlcTask Inputs/PRG_SL2L0_POWER.fbSL2L0.RTD_Bottom_1.bOverrange <-> RTD Inputs Channel 1/Status/Overrange
//     PlcTask Inputs/PRG_SL2L0_POWER.fbSL2L0.RTD_Bottom_2.bOverrange <-> RTD Inputs Channel 2/Status/Overrange
//     PlcTask Inputs/PRG_SL2L0_POWER.fbSL2L0.RTD_Bottom_1.bUnderrange <-> RTD Inputs Channel 1/Status/Underrange
//     PlcTask Inputs/PRG_SL2L0_POWER.fbSL2L0.RTD_Bottom_2.bUnderrange <-> RTD Inputs Channel 2/Status/Underrange
//     PlcTask Inputs/PRG_SL2L0_POWER.fbSL2L0.RTD_Bottom_1.iRaw <-> RTD Inputs Channel 1/Value
//     PlcTask Inputs/PRG_SL2L0_POWER.fbSL2L0.RTD_Bottom_2.iRaw <-> RTD Inputs Channel 2/Value
//   lfe_motion Instance <-> PLC Rail (EtherCAT)/Power (EK1200)/PLC Junction 2 (EK1122)/X2 SL2L0-Power (EK1100)/SL2L0-EL3202-E9
//     PlcTask Inputs/PRG_SL2L0_POWER.fbSL2L0.RTD_South_1.bError <-> RTD Inputs Channel 1/Status/Error
//     PlcTask Inputs/PRG_SL2L0_POWER.fbSL2L0.RTD_South_2.bError <-> RTD Inputs Channel 2/Status/Error
//     PlcTask Inputs/PRG_SL2L0_POWER.fbSL2L0.RTD_South_1.bOverrange <-> RTD Inputs Channel 1/Status/Overrange
//     PlcTask Inputs/PRG_SL2L0_POWER.fbSL2L0.RTD_South_2.bOverrange <-> RTD Inputs Channel 2/Status/Overrange
//     PlcTask Inputs/PRG_SL2L0_POWER.fbSL2L0.RTD_South_1.bUnderrange <-> RTD Inputs Channel 1/Status/Underrange
//     PlcTask Inputs/PRG_SL2L0_POWER.fbSL2L0.RTD_South_2.bUnderrange <-> RTD Inputs Channel 2/Status/Underrange
//     PlcTask Inputs/PRG_SL2L0_POWER.fbSL2L0.RTD_South_1.iRaw <-> RTD Inputs Channel 1/Value
//     PlcTask Inputs/PRG_SL2L0_POWER.fbSL2L0.RTD_South_2.iRaw <-> RTD Inputs Channel 2/Value
//   lfe_motion Instance <-> PLC Rail (EtherCAT)/Power (EK1200)/PLC Junction 2 (EK1122)/X2 SL2L0-Power (EK1100)/SL2L0-EL7041-E1
//     PlcTask Inputs/Main.M45.bLimitBackwardEnable <-> STM Status/Status/Digital input 1
//     PlcTask Inputs/Main.M45.bLimitForwardEnable <-> STM Status/Status/Digital input 2
//   lfe_motion Instance <-> PLC Rail (EtherCAT)/Power (EK1200)/PLC Junction 2 (EK1122)/X2 SL2L0-Power (EK1100)/SL2L0-EL7041-E3
//     PlcTask Inputs/Main.M46.bLimitBackwardEnable <-> STM Status/Status/Digital input 2
//     PlcTask Inputs/Main.M46.bLimitForwardEnable <-> STM Status/Status/Digital input 1
//   lfe_motion Instance <-> PLC Rail (EtherCAT)/Power (EK1200)/PLC Junction 2 (EK1122)/X2 SL2L0-Power (EK1100)/SL2L0-EL7041-E5
//     PlcTask Inputs/Main.M47.bLimitBackwardEnable <-> STM Status/Status/Digital input 1
//     PlcTask Inputs/Main.M47.bLimitForwardEnable <-> STM Status/Status/Digital input 2
//   lfe_motion Instance <-> PLC Rail (EtherCAT)/Power (EK1200)/PLC Junction 2 (EK1122)/X2 SL2L0-Power (EK1100)/SL2L0-EL7041-E7
//     PlcTask Inputs/Main.M48.bLimitBackwardEnable <-> STM Status/Status/Digital input 2
//     PlcTask Inputs/Main.M48.bLimitForwardEnable <-> STM Status/Status/Digital input 1
//   lfe_motion Instance <-> PLC Rail (EtherCAT)/Power (EK1200)/PMPS_FFO
//     PlcTask Outputs/GVL.fbFastFaultOutput1.q_xFastFaultOut <-> Channel 1/Output
//     PlcTask Outputs/GVL.fbFastFaultOutput2.q_xFastFaultOut <-> Channel 2/Output
//   lfe_motion Instance <-> PLC Rail (EtherCAT)/Power (EK1200)/PMPS_PRE
//     PlcTask Inputs/GVL.rReqTrans <-> IO Inputs/SattArrayReq
//     PlcTask Inputs/PRG_3_PMPS_POST.fbArbiterIO.i_stCurrentBP <-> IO Inputs/CurrentBP
//     PlcTask Inputs/PRG_3_PMPS_POST.fbArbiterIO.xTxPDO_state <-> SYNC Inputs/TxPDO state
//     PlcTask Inputs/PRG_3_PMPS_POST.fbArbiterIO.xTxPDO_toggle <-> SYNC Inputs/TxPDO toggle
//     PlcTask Outputs/GVL.rCurTrans <-> IO Outputs/SattArrayStatus
//     PlcTask Outputs/PRG_3_PMPS_POST.fbArbiterIO.q_stRequestedBP <-> IO Outputs/RequestedBP
//   lfe_motion Instance <-> NC-Task 1 SAF/Axes/Axis 1
//     PlcTask Inputs/Main.M1.Axis.NcToPlc <-> Outputs/ToPlc
//     PlcTask Outputs/Main.M1.Axis.PlcToNc <-> Inputs/FromPlc
//   lfe_motion Instance <-> NC-Task 1 SAF/Axes/Axis 10
//     PlcTask Inputs/Main.M10.Axis.NcToPlc <-> Outputs/ToPlc
//     PlcTask Outputs/Main.M10.Axis.PlcToNc <-> Inputs/FromPlc
//   lfe_motion Instance <-> NC-Task 1 SAF/Axes/Axis 11
//     PlcTask Inputs/Main.M11.Axis.NcToPlc <-> Outputs/ToPlc
//     PlcTask Outputs/Main.M11.Axis.PlcToNc <-> Inputs/FromPlc
//   lfe_motion Instance <-> NC-Task 1 SAF/Axes/Axis 12
//     PlcTask Inputs/Main.M12.Axis.NcToPlc <-> Outputs/ToPlc
//     PlcTask Outputs/Main.M12.Axis.PlcToNc <-> Inputs/FromPlc
//   lfe_motion Instance <-> NC-Task 1 SAF/Axes/Axis 13
//     PlcTask Inputs/Main.M13.Axis.NcToPlc <-> Outputs/ToPlc
//     PlcTask Outputs/Main.M13.Axis.PlcToNc <-> Inputs/FromPlc
//   lfe_motion Instance <-> NC-Task 1 SAF/Axes/Axis 14
//     PlcTask Inputs/Main.M14.Axis.NcToPlc <-> Outputs/ToPlc
//     PlcTask Outputs/Main.M14.Axis.PlcToNc <-> Inputs/FromPlc
//   lfe_motion Instance <-> NC-Task 1 SAF/Axes/Axis 15
//     PlcTask Inputs/Main.M15.Axis.NcToPlc <-> Outputs/ToPlc
//     PlcTask Outputs/Main.M15.Axis.PlcToNc <-> Inputs/FromPlc
//   lfe_motion Instance <-> NC-Task 1 SAF/Axes/Axis 16
//     PlcTask Inputs/Main.M16.Axis.NcToPlc <-> Outputs/ToPlc
//     PlcTask Outputs/Main.M16.Axis.PlcToNc <-> Inputs/FromPlc
//   lfe_motion Instance <-> NC-Task 1 SAF/Axes/Axis 17
//     PlcTask Inputs/Main.M17.Axis.NcToPlc <-> Outputs/ToPlc
//     PlcTask Outputs/Main.M17.Axis.PlcToNc <-> Inputs/FromPlc
//   lfe_motion Instance <-> NC-Task 1 SAF/Axes/Axis 18
//     PlcTask Inputs/Main.M18.Axis.NcToPlc <-> Outputs/ToPlc
//     PlcTask Outputs/Main.M18.Axis.PlcToNc <-> Inputs/FromPlc
//   lfe_motion Instance <-> NC-Task 1 SAF/Axes/Axis 19
//     PlcTask Inputs/Main.M19.Axis.NcToPlc <-> Outputs/ToPlc
//     PlcTask Outputs/Main.M19.Axis.PlcToNc <-> Inputs/FromPlc
//   lfe_motion Instance <-> NC-Task 1 SAF/Axes/Axis 2
//     PlcTask Inputs/Main.M2.Axis.NcToPlc <-> Outputs/ToPlc
//     PlcTask Outputs/Main.M2.Axis.PlcToNc <-> Inputs/FromPlc
//   lfe_motion Instance <-> NC-Task 1 SAF/Axes/Axis 20 IM1L0-XTES-MMS
//     PlcTask Inputs/Main.M20.Axis.NcToPlc <-> Outputs/ToPlc
//     PlcTask Outputs/Main.M20.Axis.PlcToNc <-> Inputs/FromPlc
//   lfe_motion Instance <-> NC-Task 1 SAF/Axes/Axis 21 IM1L0-XTES-CLZ
//     PlcTask Inputs/Main.M21.Axis.NcToPlc <-> Outputs/ToPlc
//     PlcTask Outputs/Main.M21.Axis.PlcToNc <-> Inputs/FromPlc
//   lfe_motion Instance <-> NC-Task 1 SAF/Axes/Axis 22 IM1L0-XTES-CLF
//     PlcTask Inputs/Main.M22.Axis.NcToPlc <-> Outputs/ToPlc
//     PlcTask Outputs/Main.M22.Axis.PlcToNc <-> Inputs/FromPlc
//   lfe_motion Instance <-> NC-Task 1 SAF/Axes/Axis 23 IM1L1-PPM-MMS
//     PlcTask Inputs/Main.M23.Axis.NcToPlc <-> Outputs/ToPlc
//     PlcTask Outputs/Main.M23.Axis.PlcToNc <-> Inputs/FromPlc
//   lfe_motion Instance <-> NC-Task 1 SAF/Axes/Axis 24 IM2L0-XTES-MMS
//     PlcTask Inputs/Main.M24.Axis.NcToPlc <-> Outputs/ToPlc
//     PlcTask Outputs/Main.M24.Axis.PlcToNc <-> Inputs/FromPlc
//   lfe_motion Instance <-> NC-Task 1 SAF/Axes/Axis 25 IM2L0-XTES-CLZ
//     PlcTask Inputs/Main.M25.Axis.NcToPlc <-> Outputs/ToPlc
//     PlcTask Outputs/Main.M25.Axis.PlcToNc <-> Inputs/FromPlc
//   lfe_motion Instance <-> NC-Task 1 SAF/Axes/Axis 26 IM2L0-XTES-CLF
//     PlcTask Inputs/Main.M26.Axis.NcToPlc <-> Outputs/ToPlc
//     PlcTask Outputs/Main.M26.Axis.PlcToNc <-> Inputs/FromPlc
//   lfe_motion Instance <-> NC-Task 1 SAF/Axes/Axis 27 IM3L0-PPM-MMS
//     PlcTask Inputs/Main.M27.Axis.NcToPlc <-> Outputs/ToPlc
//     PlcTask Outputs/Main.M27.Axis.PlcToNc <-> Inputs/FromPlc
//   lfe_motion Instance <-> NC-Task 1 SAF/Axes/Axis 28 IM4L0-XTES-MMS
//     PlcTask Inputs/Main.M28.Axis.NcToPlc <-> Outputs/ToPlc
//     PlcTask Outputs/Main.M28.Axis.PlcToNc <-> Inputs/FromPlc
//   lfe_motion Instance <-> NC-Task 1 SAF/Axes/Axis 29 IM4L0-XTES-CLZ
//     PlcTask Inputs/Main.M29.Axis.NcToPlc <-> Outputs/ToPlc
//     PlcTask Outputs/Main.M29.Axis.PlcToNc <-> Inputs/FromPlc
//   lfe_motion Instance <-> NC-Task 1 SAF/Axes/Axis 3
//     PlcTask Inputs/Main.M3.Axis.NcToPlc <-> Outputs/ToPlc
//     PlcTask Outputs/Main.M3.Axis.PlcToNc <-> Inputs/FromPlc
//   lfe_motion Instance <-> NC-Task 1 SAF/Axes/Axis 30 IM4L0-XTES-CLF
//     PlcTask Inputs/Main.M30.Axis.NcToPlc <-> Outputs/ToPlc
//     PlcTask Outputs/Main.M30.Axis.PlcToNc <-> Inputs/FromPlc
//   lfe_motion Instance <-> NC-Task 1 SAF/Axes/Axis 33
//     PlcTask Inputs/Main.M33.Axis.NcToPlc <-> Outputs/ToPlc
//     PlcTask Outputs/Main.M33.Axis.PlcToNc <-> Inputs/FromPlc
//   lfe_motion Instance <-> NC-Task 1 SAF/Axes/Axis 34
//     PlcTask Inputs/Main.M34.Axis.NcToPlc <-> Outputs/ToPlc
//     PlcTask Outputs/Main.M34.Axis.PlcToNc <-> Inputs/FromPlc
//   lfe_motion Instance <-> NC-Task 1 SAF/Axes/Axis 35
//     PlcTask Inputs/Main.M35.Axis.NcToPlc <-> Outputs/ToPlc
//     PlcTask Outputs/Main.M35.Axis.PlcToNc <-> Inputs/FromPlc
//   lfe_motion Instance <-> NC-Task 1 SAF/Axes/Axis 36
//     PlcTask Inputs/Main.M36.Axis.NcToPlc <-> Outputs/ToPlc
//     PlcTask Outputs/Main.M36.Axis.PlcToNc <-> Inputs/FromPlc
//   lfe_motion Instance <-> NC-Task 1 SAF/Axes/Axis 37
//     PlcTask Inputs/Main.M37.Axis.NcToPlc <-> Outputs/ToPlc
//     PlcTask Outputs/Main.M37.Axis.PlcToNc <-> Inputs/FromPlc
//   lfe_motion Instance <-> NC-Task 1 SAF/Axes/Axis 38
//     PlcTask Inputs/Main.M38.Axis.NcToPlc <-> Outputs/ToPlc
//     PlcTask Outputs/Main.M38.Axis.PlcToNc <-> Inputs/FromPlc
//   lfe_motion Instance <-> NC-Task 1 SAF/Axes/Axis 39
//     PlcTask Inputs/Main.M39.Axis.NcToPlc <-> Outputs/ToPlc
//     PlcTask Outputs/Main.M39.Axis.PlcToNc <-> Inputs/FromPlc
//   lfe_motion Instance <-> NC-Task 1 SAF/Axes/Axis 4
//     PlcTask Inputs/Main.M4.Axis.NcToPlc <-> Outputs/ToPlc
//     PlcTask Outputs/Main.M4.Axis.PlcToNc <-> Inputs/FromPlc
//   lfe_motion Instance <-> NC-Task 1 SAF/Axes/Axis 40
//     PlcTask Inputs/Main.M40.Axis.NcToPlc <-> Outputs/ToPlc
//     PlcTask Outputs/Main.M40.Axis.PlcToNc <-> Inputs/FromPlc
//   lfe_motion Instance <-> NC-Task 1 SAF/Axes/Axis 5
//     PlcTask Inputs/Main.M5.Axis.NcToPlc <-> Outputs/ToPlc
//     PlcTask Outputs/Main.M5.Axis.PlcToNc <-> Inputs/FromPlc
//   lfe_motion Instance <-> NC-Task 1 SAF/Axes/Axis 6
//     PlcTask Inputs/Main.M6.Axis.NcToPlc <-> Outputs/ToPlc
//     PlcTask Outputs/Main.M6.Axis.PlcToNc <-> Inputs/FromPlc
//   lfe_motion Instance <-> NC-Task 1 SAF/Axes/Axis 7
//     PlcTask Inputs/Main.M7.Axis.NcToPlc <-> Outputs/ToPlc
//     PlcTask Outputs/Main.M7.Axis.PlcToNc <-> Inputs/FromPlc
//   lfe_motion Instance <-> NC-Task 1 SAF/Axes/Axis 8
//     PlcTask Inputs/Main.M8.Axis.NcToPlc <-> Outputs/ToPlc
//     PlcTask Outputs/Main.M8.Axis.PlcToNc <-> Inputs/FromPlc
//   lfe_motion Instance <-> NC-Task 1 SAF/Axes/Axis 9
//     PlcTask Inputs/Main.M9.Axis.NcToPlc <-> Outputs/ToPlc
//     PlcTask Outputs/Main.M9.Axis.PlcToNc <-> Inputs/FromPlc
//   lfe_motion Instance <-> NC-Task 1 SAF/Axes/DIODE HORIZ X
//     PlcTask Inputs/Main.M53.Axis.NcToPlc <-> Outputs/ToPlc
//     PlcTask Outputs/Main.M53.Axis.PlcToNc <-> Inputs/FromPlc
//   lfe_motion Instance <-> NC-Task 1 SAF/Axes/DIODE VERT Y
//     PlcTask Inputs/Main.M54.Axis.NcToPlc <-> Outputs/ToPlc
//     PlcTask Outputs/Main.M54.Axis.PlcToNc <-> Inputs/FromPlc
//   lfe_motion Instance <-> NC-Task 1 SAF/Axes/PF1L0-WFS-MMS-01
//     PlcTask Inputs/Main.M31.Axis.NcToPlc <-> Outputs/ToPlc
//     PlcTask Outputs/Main.M31.Axis.PlcToNc <-> Inputs/FromPlc
//   lfe_motion Instance <-> NC-Task 1 SAF/Axes/PF1L0-WFS-MMS-02
//     PlcTask Inputs/Main.M32.Axis.NcToPlc <-> Outputs/ToPlc
//     PlcTask Outputs/Main.M32.Axis.PlcToNc <-> Inputs/FromPlc
//   lfe_motion Instance <-> NC-Task 1 SAF/Axes/RETICLE HORIZ X
//     PlcTask Inputs/Main.M51.Axis.NcToPlc <-> Outputs/ToPlc
//     PlcTask Outputs/Main.M51.Axis.PlcToNc <-> Inputs/FromPlc
//   lfe_motion Instance <-> NC-Task 1 SAF/Axes/RETICLE VERT Y
//     PlcTask Inputs/Main.M52.Axis.NcToPlc <-> Outputs/ToPlc
//     PlcTask Outputs/Main.M52.Axis.PlcToNc <-> Inputs/FromPlc
//   lfe_motion Instance <-> NC-Task 1 SAF/Axes/SL1L0-BOTTOM-M41
//     PlcTask Inputs/Main.M41.Axis.NcToPlc <-> Outputs/ToPlc
//     PlcTask Outputs/Main.M41.Axis.PlcToNc <-> Inputs/FromPlc
//   lfe_motion Instance <-> NC-Task 1 SAF/Axes/SL1L0-NORTH-M44
//     PlcTask Inputs/Main.M44.Axis.NcToPlc <-> Outputs/ToPlc
//     PlcTask Outputs/Main.M44.Axis.PlcToNc <-> Inputs/FromPlc
//   lfe_motion Instance <-> NC-Task 1 SAF/Axes/SL1L0-SOUTH-M42
//     PlcTask Inputs/Main.M42.Axis.NcToPlc <-> Outputs/ToPlc
//     PlcTask Outputs/Main.M42.Axis.PlcToNc <-> Inputs/FromPlc
//   lfe_motion Instance <-> NC-Task 1 SAF/Axes/SL1L0-TOP-M43
//     PlcTask Inputs/Main.M43.Axis.NcToPlc <-> Outputs/ToPlc
//     PlcTask Outputs/Main.M43.Axis.PlcToNc <-> Inputs/FromPlc
//   lfe_motion Instance <-> NC-Task 1 SAF/Axes/SL2L0-BOTTOM-M45
//     PlcTask Inputs/Main.M45.Axis.NcToPlc <-> Outputs/ToPlc
//     PlcTask Outputs/Main.M45.Axis.PlcToNc <-> Inputs/FromPlc
//   lfe_motion Instance <-> NC-Task 1 SAF/Axes/SL2L0-NORTH-M48
//     PlcTask Inputs/Main.M48.Axis.NcToPlc <-> Outputs/ToPlc
//     PlcTask Outputs/Main.M48.Axis.PlcToNc <-> Inputs/FromPlc
//   lfe_motion Instance <-> NC-Task 1 SAF/Axes/SL2L0-SOUTH-M46
//     PlcTask Inputs/Main.M46.Axis.NcToPlc <-> Outputs/ToPlc
//     PlcTask Outputs/Main.M46.Axis.PlcToNc <-> Inputs/FromPlc
//   lfe_motion Instance <-> NC-Task 1 SAF/Axes/SL2L0-TOP-M47
//     PlcTask Inputs/Main.M47.Axis.NcToPlc <-> Outputs/ToPlc
//     PlcTask Outputs/Main.M47.Axis.PlcToNc <-> Inputs/FromPlc
//   lfe_motion Instance <-> NC-Task 1 SAF/Axes/XTAL ANGLE X
//     PlcTask Inputs/Main.M49.Axis.NcToPlc <-> Outputs/ToPlc
//     PlcTask Outputs/Main.M49.Axis.PlcToNc <-> Inputs/FromPlc
//   lfe_motion Instance <-> NC-Task 1 SAF/Axes/XTAL VERT Y
//     PlcTask Inputs/Main.M50.Axis.NcToPlc <-> Outputs/ToPlc
//     PlcTask Outputs/Main.M50.Axis.PlcToNc <-> Inputs/FromPlc

CONFIGURATION lfe_motion
    RESOURCE PLC ON TwinCAT3
        TASK PlcTask(INTERVAL := T#5ms, PRIORITY := 20);
        PROGRAM PRG_1_PlcTask WITH PlcTask : PRG_1_PlcTask;
    END_RESOURCE
END_CONFIGURATION

// ---- DUTs/DUT_SATT_Filter.TcDUT
TYPE DUT_SATT_Filter :
STRUCT
    {attribute 'pytmc' := '
        pv: MATERIAL
        io: input
        field: DESC Filter material name
    '}
    sFilterMaterial : STRING;

    {attribute 'pytmc' := '
        pv: THICKNESS
        io: input
        field: DESC Filter material thickness
        field: EGU um
    '}
    fFilterThickness_um : LREAL;

    {attribute 'pytmc' := '
        pv: TRANSMISSION
        io: input
        field: DESC Current transmission value
    '}
    fTransmission : LREAL;

END_STRUCT
END_TYPE

// ---- DUTs/ST_MPA.TcDUT
TYPE ST_MPA :
STRUCT
//    i_xInsertLS AT %I*: BOOL;
//    i_xRetractLS AT %I*: BOOL;
//    _xInsertSW : BOOL;
//    _xRetractSW : BOOL;
//    q_xInsertDO AT %Q*: BOOL;
//    q_xRetractDO AT %Q*: BOOL;
//    eState : DUT_PneumaticActuator_Position;

    //Readbacks
    {attribute 'pytmc' := '
    pv: IN
    io: i
    '}
    i_bInLS    :    BOOL;
    {attribute 'pytmc' := '
    pv: OUT
    io: i
    '}
    i_bOutLS    :    BOOL;

    //Controls
    {attribute 'pytmc' := '
    pv: INSERT_DO
    io: i
    '}
    q_bRetract    :    BOOL;
    {attribute 'pytmc' := '
    pv: RETRACT_DO
    io: i
    '}
    q_bInsert    :    BOOL;

    //Logic and supervisory
    {attribute 'pytmc' := '
    pv: ILKOK
    io: i
    '}
    bILK_OK: BOOL;
    {attribute 'pytmc' := '
    pv: INSERT_OK
    io: i
    '}
    bInsertOK    :    BOOL;
    {attribute 'pytmc' := '
    pv: RETRACT_OK
    io: i
    '}
    bRetractOK    :    BOOL;
    {attribute 'pytmc' := '
    pv: IN_CMD
    io: io
    '}

    bInsert_SW        :    BOOL;
    {attribute 'pytmc' := '
    pv: OUT_CMD
    io: io
    '}
    bRetract_SW    :    BOOL;
    {attribute 'pytmc' := '
    pv: ERROR
    io: io
    '}
    bErrorPresent : BOOL;
    {attribute 'pytmc' := '
    pv: POS_STATE
    type: mbbi
    field: ZRST RETRACTED
    field: ONST INSERTED
    field: TWST MOVING
    field: THST INVALID
    io: i
    '}

    eState    :    E_PositionState := INVALID;


END_STRUCT
END_TYPE

// ---- DUTs/E_PositionState.TcDUT
TYPE E_PositionState :
(
RETRACTED    := 0,
INSERTED    := 1,
MOVING    := 2,
INVALID :=3
);
END_TYPE

// ---- GVLs/GVL.TcGVL
{attribute 'qualified_only'}
VAR_GLOBAL
    {attribute 'pytmc' := 'pv: PLC:LFE:MOTION:ARB:01'}
    fbArbiter: FB_Arbiter(1);

    {attribute 'pytmc' := 'pv: PLC:LFE:MOTION:ARB:02'}
    fbArbiter2: FB_Arbiter(2);

    {attribute 'pytmc' := 'pv: PLC:LFE:MOTION:FFO:01'}
    {attribute 'TcLinkTo' := '.q_xFastFaultOut:=TIIB[PMPS_FFO]^Channel 1^Output'}
    fbFastFaultOutput1: FB_HardwareFFOutput := (bAutoReset := TRUE, i_sNetID := '172.21.88.66.1.1');

    {attribute 'pytmc' := 'pv: PLC:LFE:MOTION:FFO:02'}
    {attribute 'TcLinkTo' := '.q_xFastFaultOut:=TIIB[PMPS_FFO]^Channel 2^Output'}
    fbFastFaultOutput2: FB_HardwareFFOutput := (bAutoReset := TRUE, i_sNetID := '172.21.88.66.1.1');

    {attribute 'pytmc' := 'pv: PLC:LFE:MOTION:PMPS:ReqTrans'}
    rReqTrans AT %I*		: ARRAY [1..PMPS_GVL.AUX_ATTENUATORS] OF ST_PMPS_Attenuator_IO;
    {attribute 'pytmc' := 'pv: PLC:LFE:MOTION:PMPS:CurTrans'}
    rCurTrans AT %Q*		: ARRAY [1..PMPS_GVL.AUX_ATTENUATORS] OF ST_PMPS_Attenuator_IO;

    ePF1L0State: E_WFS_States;
END_VAR

// ---- GVLs/Main.TcGVL
{attribute 'qualified_only'}
VAR_GLOBAL
(*
    Only includes motor definitions for the IOC
    These are hard-coded to be Main.M#,
    but are very convenient to store in a GVL,
    hence the confusing namespace here

    This should be refactored once the IOC
    supports arbitrary ads paths for motors
*)
    // AT2L0-SOLID: 19 Axes
    {attribute 'pytmc' := 'pv: AT2L0:XTES:MMS:01'}
    {attribute 'TcLinkTo' := '.bLimitForwardEnable  := TIIB[AT2L0-EL7041-01]^STM Status^Status^Digital input 2;
                              .bLimitBackwardEnable := TIIB[AT2L0-EL7041-01]^STM Status^Status^Digital input 1
    '}
    M1: ST_MotionStage := (sName := 'AT2L0:XTES:MMS:01');
    {attribute 'pytmc' := 'pv: AT2L0:XTES:MMS:02'}
    {attribute 'TcLinkTo' := '.bLimitForwardEnable  := TIIB[AT2L0-EL7041-02]^STM Status^Status^Digital input 2;
                              .bLimitBackwardEnable := TIIB[AT2L0-EL7041-02]^STM Status^Status^Digital input 1
    '}
    M2: ST_MotionStage := (sName := 'AT2L0:XTES:MMS:02');
    {attribute 'pytmc' := 'pv: AT2L0:XTES:MMS:03'}
    {attribute 'TcLinkTo' := '.bLimitForwardEnable  := TIIB[AT2L0-EL7041-03]^STM Status^Status^Digital input 2;
                              .bLimitBackwardEnable := TIIB[AT2L0-EL7041-03]^STM Status^Status^Digital input 1
    '}
    M3: ST_MotionStage := (sName := 'AT2L0:XTES:MMS:03');
    {attribute 'pytmc' := 'pv: AT2L0:XTES:MMS:04'}
    {attribute 'TcLinkTo' := '.bLimitForwardEnable  := TIIB[AT2L0-EL7041-04]^STM Status^Status^Digital input 2;
                              .bLimitBackwardEnable := TIIB[AT2L0-EL7041-04]^STM Status^Status^Digital input 1
    '}
    M4: ST_MotionStage := (sName := 'AT2L0:XTES:MMS:04');
    {attribute 'pytmc' := 'pv: AT2L0:XTES:MMS:05'}
    {attribute 'TcLinkTo' := '.bLimitForwardEnable  := TIIB[AT2L0-EL7041-05]^STM Status^Status^Digital input 2;
                              .bLimitBackwardEnable := TIIB[AT2L0-EL7041-05]^STM Status^Status^Digital input 1
    '}
    M5: ST_MotionStage := (sName := 'AT2L0:XTES:MMS:05');
    {attribute 'pytmc' := 'pv: AT2L0:XTES:MMS:06'}
    {attribute 'TcLinkTo' := '.bLimitForwardEnable  := TIIB[AT2L0-EL7041-06]^STM Status^Status^Digital input 2;
                              .bLimitBackwardEnable := TIIB[AT2L0-EL7041-06]^STM Status^Status^Digital input 1
    '}
    M6: ST_MotionStage := (sName := 'AT2L0:XTES:MMS:06');
    {attribute 'pytmc' := 'pv: AT2L0:XTES:MMS:07'}
    {attribute 'TcLinkTo' := '.bLimitForwardEnable  := TIIB[AT2L0-EL7041-07]^STM Status^Status^Digital input 2;
                              .bLimitBackwardEnable := TIIB[AT2L0-EL7041-07]^STM Status^Status^Digital input 1
    '}
    M7: ST_MotionStage := (sName := 'AT2L0:XTES:MMS:07');
    {attribute 'pytmc' := 'pv: AT2L0:XTES:MMS:08'}
    {attribute 'TcLinkTo' := '.bLimitForwardEnable  := TIIB[AT2L0-EL7041-08]^STM Status^Status^Digital input 2;
                              .bLimitBackwardEnable := TIIB[AT2L0-EL7041-08]^STM Status^Status^Digital input 1
    '}
    M8: ST_MotionStage := (sName := 'AT2L0:XTES:MMS:08');
    {attribute 'pytmc' := 'pv: AT2L0:XTES:MMS:09'}
    {attribute 'TcLinkTo' := '.bLimitForwardEnable  := TIIB[AT2L0-EL7041-09]^STM Status^Status^Digital input 2;
                              .bLimitBackwardEnable := TIIB[AT2L0-EL7041-09]^STM Status^Status^Digital input 1
    '}
    M9: ST_MotionStage := (sName := 'AT2L0:XTES:MMS:09');
    {attribute 'pytmc' := 'pv: AT2L0:XTES:MMS:10'}
    {attribute 'TcLinkTo' := '.bLimitForwardEnable  := TIIB[AT2L0-EL7041-10]^STM Status^Status^Digital input 2;
                              .bLimitBackwardEnable := TIIB[AT2L0-EL7041-10]^STM Status^Status^Digital input 1
    '}
    M10: ST_MotionStage := (sName := 'AT2L0:XTES:MMS:10');
    {attribute 'pytmc' := 'pv: AT2L0:XTES:MMS:11'}
    {attribute 'TcLinkTo' := '.bLimitForwardEnable  := TIIB[AT2L0-EL7041-11]^STM Status^Status^Digital input 2;
                              .bLimitBackwardEnable := TIIB[AT2L0-EL7041-11]^STM Status^Status^Digital input 1
    '}
    M11: ST_MotionStage := (sName := 'AT2L0:XTES:MMS:11');
    {attribute 'pytmc' := 'pv: AT2L0:XTES:MMS:12'}
    {attribute 'TcLinkTo' := '.bLimitForwardEnable  := TIIB[AT2L0-EL7041-12]^STM Status^Status^Digital input 2;
                              .bLimitBackwardEnable := TIIB[AT2L0-EL7041-12]^STM Status^Status^Digital input 1
    '}
    M12: ST_MotionStage := (sName := 'AT2L0:XTES:MMS:12');
    {attribute 'pytmc' := 'pv: AT2L0:XTES:MMS:13'}
    {attribute 'TcLinkTo' := '.bLimitForwardEnable  := TIIB[AT2L0-EL7041-13]^STM Status^Status^Digital input 2;
                              .bLimitBackwardEnable := TIIB[AT2L0-EL7041-13]^STM Status^Status^Digital input 1
    '}
    M13: ST_MotionStage := (sName := 'AT2L0:XTES:MMS:13');
    {attribute 'pytmc' := 'pv: AT2L0:XTES:MMS:14'}
    {attribute 'TcLinkTo' := '.bLimitForwardEnable  := TIIB[AT2L0-EL7041-14]^STM Status^Status^Digital input 2;
                              .bLimitBackwardEnable := TIIB[AT2L0-EL7041-14]^STM Status^Status^Digital input 1
    '}
    M14: ST_MotionStage := (sName := 'AT2L0:XTES:MMS:14');
    {attribute 'pytmc' := 'pv: AT2L0:XTES:MMS:15'}
    {attribute 'TcLinkTo' := '.bLimitForwardEnable  := TIIB[AT2L0-EL7041-15]^STM Status^Status^Digital input 2;
                              .bLimitBackwardEnable := TIIB[AT2L0-EL7041-15]^STM Status^Status^Digital input 1
    '}
    M15: ST_MotionStage := (sName := 'AT2L0:XTES:MMS:15');
    {attribute 'pytmc' := 'pv: AT2L0:XTES:MMS:16'}
    {attribute 'TcLinkTo' := '.bLimitForwardEnable  := TIIB[AT2L0-EL7041-16]^STM Status^Status^Digital input 2;
                              .bLimitBackwardEnable := TIIB[AT2L0-EL7041-16]^STM Status^Status^Digital input 1
    '}
    M16: ST_MotionStage := (sName := 'AT2L0:XTES:MMS:16');
    {attribute 'pytmc' := 'pv: AT2L0:XTES:MMS:17'}
    {attribute 'TcLinkTo' := '.bLimitForwardEnable  := TIIB[AT2L0-EL7041-17]^STM Status^Status^Digital input 2;
                              .bLimitBackwardEnable := TIIB[AT2L0-EL7041-17]^STM Status^Status^Digital input 1
    '}
    M17: ST_MotionStage := (sName := 'AT2L0:XTES:MMS:17');
    {attribute 'pytmc' := 'pv: AT2L0:XTES:MMS:18'}
    {attribute 'TcLinkTo' := '.bLimitForwardEnable  := TIIB[AT2L0-EL7041-18]^STM Status^Status^Digital input 2;
                              .bLimitBackwardEnable := TIIB[AT2L0-EL7041-18]^STM Status^Status^Digital input 1
    '}
    M18: ST_MotionStage := (sName := 'AT2L0:XTES:MMS:18');
    {attribute 'pytmc' := 'pv: AT2L0:XTES:MMS:19'}
    {attribute 'TcLinkTo' := '.bLimitForwardEnable  := TIIB[AT2L0-EL7041-19]^STM Status^Status^Digital input 2;
                              .bLimitBackwardEnable := TIIB[AT2L0-EL7041-19]^STM Status^Status^Digital input 1
    '}
    M19: ST_MotionStage := (sName := 'AT2L0:XTES:MMS:19');

    // IM1L0-XTES: 3 Axes
    {attribute 'pytmc' := 'pv: IM1L0:XTES:MMS'}
    {attribute 'TcLinkTo' := '.bLimitForwardEnable  := TIIB[IM1L0-EL7041]^STM Status^Status^Digital input 1;
                              .bBrakeRelease        := TIIB[IM1L0-EL2004]^Channel 1^Output'}
    M20: ST_MotionStage := (sName := 'IM1L0:XTES:MMS');
    {attribute 'pytmc' := 'pv: IM1L0:XTES:CLZ'}
    {attribute 'TcLinkTo' := '.bHome := TIIB[IM1L0-EL1088]^Channel 2^Input'}
    M21: ST_MotionStage := (sName := 'IM1L0:XTES:CLZ');
    {attribute 'pytmc' := 'pv: IM1L0:XTES:CLF'}
    {attribute 'TcLinkTo' := '.bHome := TIIB[IM1L0-EL1088]^Channel 4^Input'}
    M22: ST_MotionStage := (sName := 'IM1L0:XTES:CLF');

    // IM1L1-PPM: 1 Axis
    {attribute 'pytmc' := 'pv: IM1L1:PPM:MMS'}
    {attribute 'TcLinkTo' := '.bLimitForwardEnable  := TIIB[IM1L1-EL7041]^STM Status^Status^Digital input 1;
                              .bLimitBackwardEnable := TIIB[IM1L1-EL7041]^STM Status^Status^Digital input 2;
                              .bBrakeRelease        := TIIB[IM1L1-EL2004]^Channel 1^Output'}
    M23: ST_MotionStage := (sName := 'IM1L1:PPM:MMS');

    // IM2L0-XTES: 3 Axes
    {attribute 'pytmc' := 'pv: IM2L0:XTES:MMS'}
    {attribute 'TcLinkTo' := '.bBrakeRelease        := TIIB[IM2L0-EL2004]^Channel 1^Output'}
    M24: ST_MotionStage := (sName := 'IM2L0:XTES:MMS');
    {attribute 'pytmc' := 'pv: IM2L0:XTES:CLZ'}
    {attribute 'TcLinkTo' := '.bHome := TIIB[IM2L0-EL1088]^Channel 2^Input'}
    M25: ST_MotionStage := (sName := 'IM2L0:XTES:CLZ');
    {attribute 'pytmc' := 'pv: IM2L0:XTES:CLF'}
    {attribute 'TcLinkTo' := '.bHome := TIIB[IM2L0-EL1088]^Channel 4^Input'}
    M26: ST_MotionStage := (sName := 'IM2L0:XTES:CLF');

    // IM3L0-PPM: 1 Axes
    {attribute 'pytmc' := 'pv: IM3L0:PPM:MMS'}
    {attribute 'TcLinkTo' := '.bLimitForwardEnable  := TIIB[IM3L0-EL7041]^STM Status^Status^Digital input 1;
                              .bLimitBackwardEnable := TIIB[IM3L0-EL7041]^STM Status^Status^Digital input 2;
                              .bBrakeRelease        := TIIB[IM3L0-EL2004]^Channel 1^Output'}
    M27: ST_MotionStage := (sName := 'IM3L0:PPM:MMS');

    // IM4L0-XTES: 3 Axes
    {attribute 'pytmc' := 'pv: IM4L0:XTES:MMS'}

    {attribute 'TcLinkTo' := '.bLimitForwardEnable  := TIIB[IM4L0-EL7041]^STM Status^Status^Digital input 1;
                              .bBrakeRelease        := TIIB[IM4L0-EL2004]^Channel 1^Output'}
    M28: ST_MotionStage := (sName := 'IM4L0:XTES:MMS');
    {attribute 'pytmc' := 'pv: IM4L0:XTES:CLZ'}
    {attribute 'TcLinkTo' := '.bHome := TIIB[IM4L0-EL1088]^Channel 2^Input'}
    M29: ST_MotionStage := (sName := 'IM4L0:XTES:CLZ');
    {attribute 'pytmc' := 'pv: IM4L0:XTES:CLF'}
    {attribute 'TcLinkTo' := '.bHome := TIIB[IM4L0-EL1088]^Channel 4^Input'}
    M30: ST_MotionStage := (sName := 'IM4L0:XTES:CLF');

    // PF1L0-WFS: 2 Axes
    {attribute 'pytmc' := 'pv: PF1L0:WFS:MMS:Y'}
    {attribute 'TcLinkTo' := '.bLimitForwardEnable  := TIIB[PF1L0-EL7041-01]^STM Status^Status^Digital input 1;
                              .bLimitBackwardEnable := TIIB[PF1L0-EL7041-01]^STM Status^Status^Digital input 2;
                              .bBrakeRelease        := TIIB[PF1L0-EL2004]^Channel 1^Output;
                              .nRawEncoderULINT     := TIIB[PF1L0-EL5042]^FB Inputs Channel 2^Position'}
    M31: ST_MotionStage := (sName := 'PF1L0:WFS:MMS:01');
    {attribute 'pytmc' := 'pv: PF1L0:WFS:MMS:Z'}
    {attribute 'TcLinkTo' := '.nRawEncoderULINT     := TIIB[PF1L0-EL5042]^FB Inputs Channel 1^Position'}
    M32: ST_MotionStage := (sName := 'PF1L0:WFS:MMS:02');

    // RTDSL0: 8 Axes
    {attribute 'pytmc' := 'pv: RTDSL0:DIODE:MMS:01'}
    {attribute 'TcLinkTo' := '.bLimitForwardEnable  := TIIB[RTDSL0-EL7041-01]^STM Status^Status^Digital input 1;
                              .bLimitBackwardEnable := TIIB[RTDSL0-EL7041-01]^STM Status^Status^Digital input 2'}
    M33: ST_MotionStage := (sName := 'RTDSL0:DIODE:MMS:01');
    M34: ST_MotionStage;
    M35: ST_MotionStage;
    M36: ST_MotionStage;
    M37: ST_MotionStage;
    //to be uncommented when the mccallister stage on RTDSK0 is moved to RTDSLo
    (*
    {attribute 'pytmc' := 'pv: RTDSL0:SCRP:MMS:01'}
    {attribute 'TcLinkTo' := '.bLimitForwardEnable  := TIIB[RTDSL0-EL7041-02]^STM Status^Status^Digital input 1;
                              .bLimitBackwardEnable := TIIB[RTDSL0-EL7041-02]^STM Status^Status^Digital input 2'}
    M34: ST_MotionStage := (sName := 'RTDSL0:SCRP:MMS:01');
    {attribute 'pytmc' := 'pv: RTDSL0:SCRP:MMS:02'}
    {attribute 'TcLinkTo' := '.bLimitForwardEnable  := TIIB[RTDSL0-EL7041-03]^STM Status^Status^Digital input 1;
                              .bLimitBackwardEnable := TIIB[RTDSL0-EL7041-03]^STM Status^Status^Digital input 2'}
    M35: ST_MotionStage := (sName := 'RTDSL0:SCRP:MMS:02');
    {attribute 'pytmc' := 'pv: RTDSL0:SCRP:MMS:03'}
    {attribute 'TcLinkTo' := '.bLimitForwardEnable  := TIIB[RTDSL0-EL7041-04]^STM Status^Status^Digital input 1;
                              .bLimitBackwardEnable := TIIB[RTDSL0-EL7041-04]^STM Status^Status^Digital input 2'}
    M36: ST_MotionStage := (sName := 'RTDSL0:SCRP:MMS:03');
    *)
    //LDM on RTDSL0
    {attribute 'pytmc' := 'pv: RTDSL0:LDM:MMS:01'}
    {attribute 'TcLinkTo' := '.bLimitForwardEnable  := TIIB[RTDSL0-EL7041-05]^STM Status^Status^Digital input 1;
                              .bLimitBackwardEnable := TIIB[RTDSL0-EL7041-05]^STM Status^Status^Digital input 2;
                               .nRawEncoderINT := TIIB[Term 113 (EL3054)]^AI Standard Channel 1^Value'}
    //M37: ST_MotionStage := (sName := 'RTDSL0:LDM:MMS:01');
    M38: ST_MotionStage;
    M39: ST_MotionStage;
    M40: ST_MotionStage;

    // to be uncommented when mccallister stage is moved from RTDSK0 -> RTDSL0
    (*
    {attribute 'pytmc' := 'pv: RTDSL0:SCRP:LED:01'}
    {attribute 'TcLinkTo' := '.bLimitForwardEnable  := TIIB[RTDSK0-EL7041-04]^STM Status^Status^Digital input 1;
                              .bLimitBackwardEnable := TIIB[RTDSK0-EL7041-04]^STM Status^Status^Digital input 2'}
    LED1: ENUM_XPIM_States;
    *)


    // SL1L0-POWER: 4 Axes
    {attribute 'pytmc' := 'pv: SL1L0:POWER:MMS:BOTTOM'}
    {attribute 'TcLinkTo' := '.bLimitForwardEnable  := TIIB[SL1L0-EL7041-E1]^STM Status^Status^Digital input 2;
                              .bLimitBackwardEnable := TIIB[SL1L0-EL7041-E1]^STM Status^Status^Digital input 1'}
    M41: ST_MotionStage := (sName := 'SL1L0:POWER:MMS:BOTTOM');
        {attribute 'pytmc' := 'pv: SL1L0:POWER:MMS:SOUTH'}
    {attribute 'TcLinkTo' := '.bLimitForwardEnable  := TIIB[SL1L0-EL7041-E3]^STM Status^Status^Digital input 1;
                              .bLimitBackwardEnable := TIIB[SL1L0-EL7041-E3]^STM Status^Status^Digital input 2'}
    M42: ST_MotionStage := (sName := 'SL1L0:POWER:MMS:SOUTH');
    {attribute 'pytmc' := 'pv: SL1L0:POWER:MMS:TOP'}
    {attribute 'TcLinkTo' := '.bLimitForwardEnable  := TIIB[SL1L0-EL7041-E5]^STM Status^Status^Digital input 2;
                              .bLimitBackwardEnable := TIIB[SL1L0-EL7041-E5]^STM Status^Status^Digital input 1'}
    M43: ST_MotionStage := (sName := 'SL1L0:POWER:MMS:TOP');
    {attribute 'pytmc' := 'pv: SL1L0:POWER:MMS:NORTH'}
    {attribute 'TcLinkTo' := '.bLimitForwardEnable  := TIIB[SL1L0-EL7041-E7]^STM Status^Status^Digital input 1;
                              .bLimitBackwardEnable := TIIB[SL1L0-EL7041-E7]^STM Status^Status^Digital input 2'}
    M44: ST_MotionStage := (sName := 'SL1L0:POWER:MMS:NORTH');

    // SL2L0-POWER: 4 Axes
    {attribute 'pytmc' := 'pv: SL2L0:POWER:MMS:BOTTOM'}
    {attribute 'TcLinkTo' := '.bLimitForwardEnable  := TIIB[SL2L0-EL7041-E1]^STM Status^Status^Digital input 2;
                              .bLimitBackwardEnable := TIIB[SL2L0-EL7041-E1]^STM Status^Status^Digital input 1'}
    M45: ST_MotionStage := (sName := 'SL2L0:POWER:MMS:BOTTOM');
    {attribute 'pytmc' := 'pv: SL2L0:POWER:MMS:SOUTH'}
    {attribute 'TcLinkTo' := '.bLimitForwardEnable  := TIIB[SL2L0-EL7041-E3]^STM Status^Status^Digital input 1;
                              .bLimitBackwardEnable := TIIB[SL2L0-EL7041-E3]^STM Status^Status^Digital input 2'}
    M46: ST_MotionStage := (sName := 'SL2L0:POWER:MMS:SOUTH');
    {attribute 'pytmc' := 'pv: SL2L0:POWER:MMS:TOP'}
    {attribute 'TcLinkTo' := '.bLimitForwardEnable  := TIIB[SL2L0-EL7041-E5]^STM Status^Status^Digital input 2;
                              .bLimitBackwardEnable := TIIB[SL2L0-EL7041-E5]^STM Status^Status^Digital input 1'}
    M47: ST_MotionStage := (sName := 'SL2L0:POWER:MMS:TOP');
    {attribute 'pytmc' := 'pv: SL2L0:POWER:MMS:NORTH'}
    {attribute 'TcLinkTo' := '.bLimitForwardEnable  := TIIB[SL2L0-EL7041-E7]^STM Status^Status^Digital input 1;
                              .bLimitBackwardEnable := TIIB[SL2L0-EL7041-E7]^STM Status^Status^Digital input 2'}
    M48: ST_MotionStage := (sName := 'SL2L0:POWER:MMS:NORTH');

    // SP1L0-KMONO: 6 Axes
    {attribute 'pytmc' := 'pv: SP1L0:KMONO:MMS:XTAL_ANGLE'}
    M49: ST_MotionStage := (sName := 'SP1L0:KMONO:MMS:XTAL_ANGLE');
    {attribute 'pytmc' := 'pv: SP1L0:KMONO:MMS:XTAL_VERT'}
    //{attribute 'TcLinkTo' := '.bLimitForwardEnable  := TIIB[SP1L0-EL7041-E2-MOTORS]^STM Status^Status^Digital input 2;
    //                          .bLimitBackwardEnable := TIIB[SP1L0-EL7041-E2-MOTORS]^STM Status^Status^Digital input 1'}
    M50: ST_MotionStage := (sName := 'SP1L0:KMONO:MMS:XTAL_VERT');
    {attribute 'pytmc' := 'pv: SP1L0:KMONO:MMS:RET_HORIZ'}
    //{attribute 'TcLinkTo' := '.bLimitForwardEnable  := TIIB[SP1L0-EL7041-E3-MOTORS]^STM Status^Status^Digital input 2;
    //                          .bLimitBackwardEnable := TIIB[SP1L0-EL7041-E3-MOTORS]^STM Status^Status^Digital input 1'}
    M51: ST_MotionStage := (sName := 'SP1L0:KMONO:MMS:RET_HORIZ');
    {attribute 'pytmc' := 'pv: SP1L0:KMONO:MMS:RET_VERT'}
    //{attribute 'TcLinkTo' := '.bLimitForwardEnable  := TIIB[SP1L0-EL7041-E4-MOTORS]^STM Status^Status^Digital input 1;
    //                          .bLimitBackwardEnable := TIIB[SP1L0-EL7041-E4-MOTORS]^STM Status^Status^Digital input 2'}
    M52: ST_MotionStage := (sName := 'SP1L0:KMONO:MMS:RET_VERT');
    {attribute 'pytmc' := 'pv: SP1L0:KMONO:MMS:DIODE_HORIZ'}
    //{attribute 'TcLinkTo' := '.bLimitForwardEnable  := TIIB[SP1L0-EL7041-E5-MOTORS]^STM Status^Status^Digital input 2;
    //                          .bLimitBackwardEnable := TIIB[SP1L0-EL7041-E5-MOTORS]^STM Status^Status^Digital input 1'}
    M53: ST_MotionStage := (sName := 'SP1L0:KMONO:MMS:DIODE_HORIZ');
    {attribute 'pytmc' := 'pv: SP1L0:KMONO:MMS:DIODE_VERT'}
    //{attribute 'TcLinkTo' := '.bLimitForwardEnable  := TIIB[SP1L0-EL7041-E6-MOTORS]^STM Status^Status^Digital input 1;
    //                          .bLimitBackwardEnable := TIIB[SP1L0-EL7041-E6-MOTORS]^STM Status^Status^Digital input 2'}
    M54: ST_MotionStage := (sName := 'SP1L0:KMONO:MMS:DIODE_VERT');

        // Three_Stage_RTDSX0: 3 Axes
     (*   to uncomment when stage is moved to RTDSL0
    {attribute 'pytmc' := 'pv: RTDSX0:MMS:01'}
    {attribute 'TcLinkTo' := '.bLimitForwardEnable  := TIIB[SP1L0-EL7041-E2-MOTORS]^STM Status^Status^Digital input 2;
                              .bLimitBackwardEnable := TIIB[SP1L0-EL7041-E2-MOTORS]^STM Status^Status^Digital input 1'}
    M55: ST_MotionStage := (sName := 'RTDSX0:MMS:01');

     {attribute 'pytmc' := 'pv: RTDSX0:MMS:02'}
    {attribute 'TcLinkTo' := '.bLimitForwardEnable  := TIIB[SP1L0-EL7041-E2-MOTORS]^STM Status^Status^Digital input 2;
                              .bLimitBackwardEnable := TIIB[SP1L0-EL7041-E2-MOTORS]^STM Status^Status^Digital input 1'}
    M56: ST_MotionStage := (sName := 'RTDSX0:MMS:02');

    {attribute 'pytmc' := 'pv: RTDSX0:MMS:03'}
    {attribute 'TcLinkTo' := '.bLimitForwardEnable  := TIIB[SP1L0-EL7041-E2-MOTORS]^STM Status^Status^Digital input 2;
                              .bLimitBackwardEnable := TIIB[SP1L0-EL7041-E2-MOTORS]^STM Status^Status^Digital input 1'}
    M57: ST_MotionStage := (sName := 'RTDSX0:MMS:03');
    *)
END_VAR

// ---- GVLs/RTDSL0.TcGVL
//{attribute 'qualified_only'}
VAR_GLOBAL
    {attribute 'pytmc' :=' pv: RTDSL0:MPA:01 '}
    RTDSL0_MPA_01: FB_MPA := (sName := 'RTDSL0:MPA:01');

    {attribute 'pytmc' :=' pv: RTDSL0:MPA:02 '}
    RTDSL0_MPA_02: FB_MPA := (sName := 'RTDSL0:MPA:02');

    {attribute 'pytmc' :=' pv: RTDSL0:MPA:03 '}
    RTDSL0_MPA_03: FB_MPA := (sName := 'RTDSL0:MPA:03');

    {attribute 'pytmc' :=' pv: RTDSL0:MPA:04 '}
    RTDSL0_MPA_04: FB_MPA := (sName := 'RTDSL0:MPA:04');


END_VAR

// ---- Version/Global_Version.TcGVL
{attribute 'TcGenerated'}
{attribute 'no-analysis'}
{attribute 'linkalways'}
// This function has been automatically generated from the project information.
VAR_GLOBAL CONSTANT
    {attribute 'const_non_replaced'}
    stLibVersion_lcls_plc_lfe_motion : ST_LibVersion := (iMajor := 0, iMinor := 0, iBuild := 0, iRevision := 0, nFlags := 0, sVersion := '0.0.0');
END_VAR

// ---- POUs/PRG_1_PlcTask.TcPOU
PROGRAM PRG_1_PlcTask
(*
    Launch site for each component's program
    Only "fast" programs are allowed here,
    anything else needs to be relegated to a second task
*)

PRG_2_PMPS_PRE();

PRG_AT2L0_SOLID();
PRG_IM1L0_XTES();
PRG_IM1L1_PPM();
PRG_IM2L0_XTES();
PRG_IM3L0_PPM();
PRG_IM4L0_XTES();
PRG_PF1L0_WFS();
PRG_RTDSL0();
PRG_SL1L0_POWER();
PRG_SL2L0_POWER();
//PRG_SP1L0_KMONO();

PRG_3_PMPS_POST();
PRG_4_LOG();

END_PROGRAM

// ---- POUs/PRG_2_PMPS_PRE.TcPOU
PROGRAM PRG_2_PMPS_PRE
VAR

END_VAR


MOTION_GVL.fbStandardPMPSDB(
    io_fbFFHWO:=GVL.fbFastFaultOutput1,
    bEnable:=TRUE,
    sPLCName:='plc-lfe-motion',
);

END_PROGRAM

// ---- POUs/PRG_AT2L0_SOLID.TcPOU
PROGRAM PRG_AT2L0_SOLID
VAR
    bAT2L0_debug: BOOL := FALSE;
    nAT2L0_enableMode: ENUM_StageEnableMode := ENUM_StageEnableMode.DURING_MOTION;

    iIndex: INT;
    fbAT2L0_motion: ARRAY [1..19] OF FB_MotionStage;
    fbAT2L0_axes: ARRAY [1..19] OF POINTER TO DUT_MotionStage;
    fbAT2L0_ffo: ARRAY[1..19] OF FB_AttFFO;

    {attribute 'pytmc' := '
        pv: AT2L0:XTES:MMS
        expand: :%.2d:FILTER
    '}
    fbAT2L0_filters: ARRAY[1..19] OF DUT_SATT_Filter;

    {attribute 'pytmc' := '
        pv: AT2L0:XTES:TRANSMISSION
        field: DESC Overall transmission of AT2L0
    '}
    fTransmission: LREAL;

    {attribute 'pytmc' := '
        pv: AT2L0:XTES:MMS
        expand: :%.2d:STATE
    '}
    fbAT2L0_states: ARRAY[1..19] OF FB_PositionState1D_InOut;

    stOut: ST_PositionState  := (
        fPosition := 24,
        fDelta := 2,
        fVelocity := 6,
        bMoveOk := TRUE,
        bValid := TRUE);

    stIn: ST_PositionState  := (
        fPosition := 0,
        fDelta := 2,
        fVelocity := 6,
        bMoveOk := TRUE,
        bValid := TRUE);

    // For plotting voltage/current during debugging
    nM1CoilARaw AT %I*: UINT;
    nM1CoilBRaw AT %I*: UINT; // ..CoilBRaw is currently linked to EL7041 'Coil Voltage A'
    nM1CoilA: INT;
    nM1CoilB: INT;
    //nM1Current: INT;
    nM2CoilARaw AT %I*: UINT;
    nM2CoilBRaw AT %I*: UINT;
    nM2CoilA: INT;
    nM2CoilB: INT;
    //nM2Current: INT;
    nM3CoilARaw AT %I*: UINT;
    nM3CoilBRaw AT %I*: UINT;
    nM3CoilA: INT;
    nM3CoilB: INT;
    //nM3Current: INT;
    nM4CoilARaw AT %I*: UINT;
    nM4CoilBRaw AT %I*: UINT;
    nM4CoilA: INT;
    nM4CoilB: INT;
    //nM4Current: INT;
    nM5CoilARaw AT %I*: UINT;
    nM5CoilBRaw AT %I*: UINT;
    nM5CoilA: INT;
    nM5CoilB: INT;
    //nM5Current: INT;
    nM6CoilARaw AT %I*: UINT;
    nM6CoilBRaw AT %I*: UINT;
    nM6CoilA: INT;
    nM6CoilB: INT;
    //nM6Current: INT;
    nM7CoilARaw AT %I*: UINT;
    nM7CoilBRaw AT %I*: UINT;
    nM7CoilA: INT;
    nM7CoilB: INT;
    //nM7Current: INT;
    nM8CoilARaw AT %I*: UINT;
    nM8CoilBRaw AT %I*: UINT;
    nM8CoilA: INT;
    nM8CoilB: INT;
    //nM8Current: INT;
    nM9CoilARaw AT %I*: UINT;
    nM9CoilBRaw AT %I*: UINT;
    nM9CoilA: INT;
    nM9CoilB: INT;
    //nM9Current: INT;
    nM10CoilARaw AT %I*: UINT;
    nM10CoilBRaw AT %I*: UINT;
    nM10CoilA: INT;
    nM10CoilB: INT;
    //nM10Current: INT;
    nM11CoilARaw AT %I*: UINT;
    nM11CoilBRaw AT %I*: UINT;
    nM11CoilA: INT;
    nM11CoilB: INT;
    //nM11Current: INT;
    nM12CoilARaw AT %I*: UINT;
    nM12CoilBRaw AT %I*: UINT;
    nM12CoilA: INT;
    nM12CoilB: INT;
    //nM12Current: INT;
    nM13CoilARaw AT %I*: UINT;
    nM13CoilBRaw AT %I*: UINT;
    nM13CoilA: INT;
    nM13CoilB: INT;
    //nM13Current: INT;
    nM14CoilARaw AT %I*: UINT;
    nM14CoilBRaw AT %I*: UINT;
    nM14CoilA: INT;
    nM14CoilB: INT;
    //nM14Current: INT;
    nM15CoilARaw AT %I*: UINT;
    nM15CoilBRaw AT %I*: UINT;
    nM15CoilA: INT;
    nM15CoilB: INT;
    //nM15Current: INT;
    nM16CoilARaw AT %I*: UINT;
    nM16CoilBRaw AT %I*: UINT;
    nM16CoilA: INT;
    nM16CoilB: INT;
    //nM16Current: INT;
    nM17CoilARaw AT %I*: UINT;
    nM17CoilBRaw AT %I*: UINT;
    nM17CoilA: INT;
    nM17CoilB: INT;
    //nM17Current: INT;
    nM18CoilARaw AT %I*: UINT;
    nM18CoilBRaw AT %I*: UINT;
    nM18CoilA: INT;
    nM18CoilB: INT;
    //nM18Current: INT;
    nM19CoilARaw AT %I*: UINT;
    nM19CoilBRaw AT %I*: UINT;
    nM19CoilA: INT;
    nM19CoilB: INT;
    //nM19Current: INT;

    stFilter : REFERENCE TO DUT_SATT_Filter;
    fFilterDensity : LREAL;
    fFilterAtomicMass : LREAL;
    fbAtomicMass : FB_AtomicMass;
    fbAttenuatorElementDensity : FB_AttenuatorElementDensity;
    fAbsorptionConstant : LREAL;
    bError : BOOL;

END_VAR


fbAT2L0_axes[1]:= ADR(Main.M1);
fbAT2L0_axes[2]:= ADR(Main.M2);
fbAT2L0_axes[3]:= ADR(Main.M3);
fbAT2L0_axes[4]:= ADR(Main.M4);
fbAT2L0_axes[5]:= ADR(Main.M5);
fbAT2L0_axes[6]:= ADR(Main.M6);
fbAT2L0_axes[7]:= ADR(Main.M7);
fbAT2L0_axes[8]:= ADR(Main.M8);
fbAT2L0_axes[9]:= ADR(Main.M9);
fbAT2L0_axes[10]:= ADR(Main.M10);
fbAT2L0_axes[11]:= ADR(Main.M11);
fbAT2L0_axes[12]:= ADR(Main.M12);
fbAT2L0_axes[13]:= ADR(Main.M13);
fbAT2L0_axes[14]:= ADR(Main.M14);
fbAT2L0_axes[15]:= ADR(Main.M15);
fbAT2L0_axes[16]:= ADR(Main.M16);
fbAT2L0_axes[17]:= ADR(Main.M17);
fbAT2L0_axes[18]:= ADR(Main.M18);
fbAT2L0_axes[19]:= ADR(Main.M19);

(* Not a filter *)
fbAT2L0_filters[ 1].fFilterThickness_um := 0;
fbAT2L0_filters[ 1].sFilterMaterial     := '';

fbAT2L0_filters[ 2].fFilterThickness_um := 1280.0;
fbAT2L0_filters[ 2].sFilterMaterial     := 'C';
fbAT2L0_filters[ 3].fFilterThickness_um := 320.0;
fbAT2L0_filters[ 3].sFilterMaterial     := 'C';
fbAT2L0_filters[ 4].fFilterThickness_um := 640.0;
fbAT2L0_filters[ 4].sFilterMaterial     := 'C';
fbAT2L0_filters[ 5].fFilterThickness_um := 160.0;
fbAT2L0_filters[ 5].sFilterMaterial     := 'C';
fbAT2L0_filters[ 6].fFilterThickness_um := 80.0;
fbAT2L0_filters[ 6].sFilterMaterial     := 'C';
fbAT2L0_filters[ 7].fFilterThickness_um := 40.0;
fbAT2L0_filters[ 7].sFilterMaterial     := 'C';
fbAT2L0_filters[ 8].fFilterThickness_um := 20.0;
fbAT2L0_filters[ 8].sFilterMaterial     := 'C';
fbAT2L0_filters[ 9].fFilterThickness_um := 10.0;
fbAT2L0_filters[ 9].sFilterMaterial     := 'C';

fbAT2L0_filters[10].fFilterThickness_um := 10240.0;
fbAT2L0_filters[10].sFilterMaterial     := 'Si';
fbAT2L0_filters[11].fFilterThickness_um := 5120.0;
fbAT2L0_filters[11].sFilterMaterial     := 'Si';
fbAT2L0_filters[12].fFilterThickness_um := 2560.0;
fbAT2L0_filters[12].sFilterMaterial     := 'Si';
fbAT2L0_filters[13].fFilterThickness_um := 1280.0;
fbAT2L0_filters[13].sFilterMaterial     := 'Si';
fbAT2L0_filters[14].fFilterThickness_um := 640.0;
fbAT2L0_filters[14].sFilterMaterial     := 'Si';
fbAT2L0_filters[15].fFilterThickness_um := 320.0;
fbAT2L0_filters[15].sFilterMaterial     := 'Si';
fbAT2L0_filters[16].fFilterThickness_um := 160.0;
fbAT2L0_filters[16].sFilterMaterial     := 'Si';
fbAT2L0_filters[17].fFilterThickness_um := 80.0;
fbAT2L0_filters[17].sFilterMaterial     := 'Si';
fbAT2L0_filters[18].fFilterThickness_um := 40.0;
fbAT2L0_filters[18].sFilterMaterial     := 'Si';
fbAT2L0_filters[19].fFilterThickness_um := 20.0;
fbAT2L0_filters[19].sFilterMaterial     := 'Si';

IF bAT2L0_debug THEN
    nAT2L0_enableMode := ENUM_StageEnableMode.ALWAYS;
ELSE
    nAT2L0_enableMode := ENUM_StageEnableMode.DURING_MOTION;
END_IF


(* Recalculate the overall transmission below *)
fTransmission := 1.0;

FOR iIndex := 1 TO 19 DO
    fbAT2L0_motion[iIndex](stMotionStage := fbAT2L0_axes[iIndex]^);
    fbAT2L0_axes[iIndex]^.nEnableMode := nAT2L0_enableMode;
    fbAT2L0_axes[iIndex]^.bHardwareEnable := TRUE;
    fbAT2L0_axes[iIndex]^.bPowerSelf := TRUE;
    stFilter REF= fbAT2L0_filters[iIndex];

    fbAT2L0_states[iIndex](
        stMotionStage := fbAT2L0_axes[iIndex]^,
        stOut := stOut,
        stIn := stIn);

    fbAT2L0_ffo[iIndex](
        stMotionStage := fbAT2L0_axes[iIndex]^,
        enumState := fbAT2L0_states[iIndex].eStateGet,
        fbFFHWO := GVL.fbFastFaultOutput1);

    IF fbAT2L0_states[iIndex].eStateGet = ENUM_EpicsInOut.UNKNOWN THEN
        stFilter.fTransmission := 0.0;
    ELSIF fbAT2L0_states[iIndex].eStateGet = ENUM_EpicsInOut.OUT OR stFilter.sFilterMaterial = '' THEN
        stFilter.fTransmission := 1.0;
    ELSE
        fbAtomicMass(sName:=stFilter.sFilterMaterial, fValue=>fFilterAtomicMass);
        fbAttenuatorElementDensity(sName:=stFilter.sFilterMaterial, fDensity=>fFilterDensity);

        fAbsorptionConstant := F_CalculateAbsorptionConstant(
            sElement:=stFilter.sFilterMaterial,
            fEnergyEV:=PMPS_GVL.stCurrentBeamParameters.neV,
            fDensity_gm3:=fFilterDensity,
            fAtomicWeight:=fFilterAtomicMass,
            bError=>bError,
        );
        stFilter.fTransmission := F_CalculateTransmission(
            fAbsorptionConstant:=fAbsorptionConstant,
            fThickness_in_m:=stFilter.fFilterThickness_um * 1.0E-6
        );
    END_IF

    fTransmission := fTransmission * stFilter.fTransmission;
END_FOR

IF fbAT2L0_states[1].eStateGet = ENUM_EpicsInOut.IN THEN
    (* Inspection mirror blocks the beam *)
    GVL.rCurTrans[PMPS.L_Attenuators.AT2L0].nTran := 0.0;
    (* TODO fast fault as well *)
ELSE
    GVL.rCurTrans[PMPS.L_Attenuators.AT2L0].nTran := LREAL_TO_REAL(fTransmission);
END_IF

iIndex := 0;

nM1CoilA := UINT_TO_INT(nM1CoilARaw);
nM1CoilB := UINT_TO_INT(nM1CoilBRaw);
//nM1Current := ABS(nM1CoilA) + ABS(nM1CoilB);
nM2CoilA := UINT_TO_INT(nM2CoilARaw);
nM2CoilB := UINT_TO_INT(nM2CoilBRaw);
//nM2Current := ABS(nM2CoilA) + ABS(nM2CoilB);
nM3CoilA := UINT_TO_INT(nM3CoilARaw);
nM3CoilB := UINT_TO_INT(nM3CoilBRaw);
//nM3Current := ABS(nM3CoilA) + ABS(nM3CoilB);
nM4CoilA := UINT_TO_INT(nM4CoilARaw);
nM4CoilB := UINT_TO_INT(nM4CoilBRaw);
//nM4Current := ABS(nM4CoilA) + ABS(nM4CoilB);
nM5CoilA := UINT_TO_INT(nM5CoilARaw);
nM5CoilB := UINT_TO_INT(nM5CoilBRaw);
//nM5Current := ABS(nM5CoilA) + ABS(nM5CoilB);
nM5CoilA := UINT_TO_INT(nM5CoilARaw);
nM5CoilB := UINT_TO_INT(nM5CoilBRaw);
//nM5Current := ABS(nM5CoilA) + ABS(nM5CoilB);
nM6CoilA := UINT_TO_INT(nM6CoilARaw);
nM6CoilB := UINT_TO_INT(nM6CoilBRaw);
//nM6Current := ABS(nM6CoilA) + ABS(nM6CoilB);
nM7CoilA := UINT_TO_INT(nM7CoilARaw);
nM7CoilB := UINT_TO_INT(nM7CoilBRaw);
//nM7Current := ABS(nM7CoilA) + ABS(nM7CoilB);
nM8CoilA := UINT_TO_INT(nM8CoilARaw);
nM8CoilB := UINT_TO_INT(nM8CoilBRaw);
//nM8Current := ABS(nM9CoilA) + ABS(nM9CoilB);
nM9CoilA := UINT_TO_INT(nM9CoilARaw);
nM9CoilB := UINT_TO_INT(nM9CoilBRaw);
//nM9Current := ABS(nM9CoilA) + ABS(nM9CoilB);
nM10CoilA := UINT_TO_INT(nM10CoilARaw);
nM10CoilB := UINT_TO_INT(nM10CoilBRaw);
//nM10Current := ABS(nM10CoilA) + ABS(nM10CoilB);
nM11CoilA := UINT_TO_INT(nM11CoilARaw);
nM11CoilB := UINT_TO_INT(nM11CoilBRaw);
//nM11Current := ABS(nM11CoilA) + ABS(nM11CoilB);
nM12CoilA := UINT_TO_INT(nM12CoilARaw);
nM12CoilB := UINT_TO_INT(nM12CoilBRaw);
//nM12Current := ABS(nM12CoilA) + ABS(nM12CoilB);
nM13CoilA := UINT_TO_INT(nM13CoilARaw);
nM13CoilB := UINT_TO_INT(nM13CoilBRaw);
//nM13Current := ABS(nM13CoilA) + ABS(nM13CoilB);
nM14CoilA := UINT_TO_INT(nM14CoilARaw);
nM14CoilB := UINT_TO_INT(nM14CoilBRaw);
//nM14Current := ABS(nM14CoilA) + ABS(nM14CoilB);
nM15CoilA := UINT_TO_INT(nM15CoilARaw);
nM15CoilB := UINT_TO_INT(nM15CoilBRaw);
//nM15Current := ABS(nM15CoilA) + ABS(nM15CoilB);
nM16CoilA := UINT_TO_INT(nM16CoilARaw);
nM16CoilB := UINT_TO_INT(nM16CoilBRaw);
//nM16Current := ABS(nM16CoilA) + ABS(nM16CoilB);
nM17CoilA := UINT_TO_INT(nM17CoilARaw);
nM17CoilB := UINT_TO_INT(nM17CoilBRaw);
//nM17Current := ABS(nM17CoilA) + ABS(nM17CoilB);
nM18CoilA := UINT_TO_INT(nM18CoilARaw);
nM18CoilB := UINT_TO_INT(nM18CoilBRaw);
//nM18Current := ABS(nM2CoilA) + ABS(nM18CoilB);
nM19CoilA := UINT_TO_INT(nM19CoilARaw);
nM19CoilB := UINT_TO_INT(nM19CoilBRaw);
//nM19Current := ABS(nM2CoilA) + ABS(nM2CoilB);

END_PROGRAM

// ---- Temp/FB_AttFFO.TcPOU
FUNCTION_BLOCK FB_AttFFO
VAR_IN_OUT
    stMotionStage: DUT_MotionStage;
    enumState: ENUM_EpicsInOut;
    fbFFHWO: FB_HardwareFFOutput;
END_VAR
VAR_OUTPUT
    bIsNotMoving: BOOL;
END_VAR
VAR
    fbFF: FB_FastFault := (i_Desc := 'Device is moving',
                           i_TypeCode := 16#2100,
                           i_xAutoReset := TRUE);
END_VAR

bIsNotMoving := NOT stMotionStage.Axis.Status.Moving;
fbFF(i_DevName := stMotionStage.sName,
     i_xOK := bIsNotMoving AND enumState <> ENUM_EpicsInOut.UNKNOWN,
     io_fbFFHWO := fbFFHWO);

END_FUNCTION_BLOCK

// ---- POUs/FB_AttenuatorElementDensity.TcPOU
FUNCTION_BLOCK FB_AttenuatorElementDensity
VAR_INPUT
    sName : STRING;
END_VAR
VAR_OUTPUT
    fDensity : LREAL;
    bFound : BOOL;
END_VAR
VAR
    fbElementDensity : FB_ElementDensity;
    fDensity_gm3 : LREAL;
END_VAR

IF sName = 'C' THEN
    (* Special-case diamond here *)
    fDensity := 3.51E6;  (* C (Diamond) g/m^3 *)
ELSE
    fbElementDensity(sName:=sName);
    IF fbElementDensity.bFound THEN
        fDensity := fbElementDensity.fValue * 1.0E6; (* g/cm^3 -> g/m^3 *)
    ELSE
        fDensity := 0.0;
    END_IF
END_IF

END_FUNCTION_BLOCK

// ---- POUs/PRG_IM1L0_XTES.TcPOU
PROGRAM PRG_IM1L0_XTES
VAR
    {attribute 'pytmc' := '
        pv: IM1L0:XTES
        io: io
    '}
    {attribute 'TcLinkTo' := '.bZoomEndFwd := TIIB[IM1L0-EL1088]^Channel 1^Input;
                              .bZoomEndBwd := TIIB[IM1L0-EL1088]^Channel 2^Input;
                              .bFocusEndFwd := TIIB[IM1L0-EL1088]^Channel 3^Input;
                              .bFocusEndBwd := TIIB[IM1L0-EL1088]^Channel 4^Input;
                              .fbOpal.bOpalPower := TIIB[IM1L0-EL2004]^Channel 2^Output;
                              .fbLED.bLedPower := TIIB[IM1L0-EL2004]^Channel 3^Output'}
    fbIM1L0: FB_XPIM;
    {attribute 'pytmc' := '
        pv: IM1L0:XTES:FLOW_OK
        field: ZNAM LOW
        field: ONAM OK
    '}
    {attribute 'TcLinkTo' := 'TIIB[IM1L0-EL7342]^DCM Status Channel 1^Status^Digital input 1'}
    bIM1L0FlowOk AT %I*: BOOL;
    {attribute 'TcLinkTo' := '.Status := TIIB[IM1L0-EL6002]^COM TxPDO-Map Inputs Channel 1^Status;
                              .D[0] := TIIB[IM1L0-EL6002]^COM TxPDO-Map Inputs Channel 1^Data In 0;
                              .D[1] := TIIB[IM1L0-EL6002]^COM TxPDO-Map Inputs Channel 1^Data In 1;
                              .D[2] := TIIB[IM1L0-EL6002]^COM TxPDO-Map Inputs Channel 1^Data In 2;
                              .D[3] := TIIB[IM1L0-EL6002]^COM TxPDO-Map Inputs Channel 1^Data In 3;
                              .D[4] := TIIB[IM1L0-EL6002]^COM TxPDO-Map Inputs Channel 1^Data In 4;
                              .D[5] := TIIB[IM1L0-EL6002]^COM TxPDO-Map Inputs Channel 1^Data In 5;
                              .D[6] := TIIB[IM1L0-EL6002]^COM TxPDO-Map Inputs Channel 1^Data In 6;
                              .D[7] := TIIB[IM1L0-EL6002]^COM TxPDO-Map Inputs Channel 1^Data In 7;
                              .D[8] := TIIB[IM1L0-EL6002]^COM TxPDO-Map Inputs Channel 1^Data In 8;
                              .D[9] := TIIB[IM1L0-EL6002]^COM TxPDO-Map Inputs Channel 1^Data In 9;
                              .D[10] := TIIB[IM1L0-EL6002]^COM TxPDO-Map Inputs Channel 1^Data In 10;
                              .D[11] := TIIB[IM1L0-EL6002]^COM TxPDO-Map Inputs Channel 1^Data In 11;
                              .D[12] := TIIB[IM1L0-EL6002]^COM TxPDO-Map Inputs Channel 1^Data In 12;
                              .D[13] := TIIB[IM1L0-EL6002]^COM TxPDO-Map Inputs Channel 1^Data In 13;
                              .D[14] := TIIB[IM1L0-EL6002]^COM TxPDO-Map Inputs Channel 1^Data In 14;
                              .D[15] := TIIB[IM1L0-EL6002]^COM TxPDO-Map Inputs Channel 1^Data In 15;
                              .D[16] := TIIB[IM1L0-EL6002]^COM TxPDO-Map Inputs Channel 1^Data In 16;
                              .D[17] := TIIB[IM1L0-EL6002]^COM TxPDO-Map Inputs Channel 1^Data In 17;
                              .D[18] := TIIB[IM1L0-EL6002]^COM TxPDO-Map Inputs Channel 1^Data In 18;
                              .D[19] := TIIB[IM1L0-EL6002]^COM TxPDO-Map Inputs Channel 1^Data In 19;
                              .D[20] := TIIB[IM1L0-EL6002]^COM TxPDO-Map Inputs Channel 1^Data In 20;
                              .D[21] := TIIB[IM1L0-EL6002]^COM TxPDO-Map Inputs Channel 1^Data In 21'}
    stEL6In AT %I*: EL6InData22b;
    {attribute 'TcLinkTo' := '.Ctrl := TIIB[IM1L0-EL6002]^COM RxPDO-Map Outputs Channel 1^Ctrl;
                              .D[0] := TIIB[IM1L0-EL6002]^COM RxPDO-Map Outputs Channel 1^Data Out 0;
                              .D[1] := TIIB[IM1L0-EL6002]^COM RxPDO-Map Outputs Channel 1^Data Out 1;
                              .D[2] := TIIB[IM1L0-EL6002]^COM RxPDO-Map Outputs Channel 1^Data Out 2;
                              .D[3] := TIIB[IM1L0-EL6002]^COM RxPDO-Map Outputs Channel 1^Data Out 3;
                              .D[4] := TIIB[IM1L0-EL6002]^COM RxPDO-Map Outputs Channel 1^Data Out 4;
                              .D[5] := TIIB[IM1L0-EL6002]^COM RxPDO-Map Outputs Channel 1^Data Out 5;
                              .D[6] := TIIB[IM1L0-EL6002]^COM RxPDO-Map Outputs Channel 1^Data Out 6;
                              .D[7] := TIIB[IM1L0-EL6002]^COM RxPDO-Map Outputs Channel 1^Data Out 7;
                              .D[8] := TIIB[IM1L0-EL6002]^COM RxPDO-Map Outputs Channel 1^Data Out 8;
                              .D[9] := TIIB[IM1L0-EL6002]^COM RxPDO-Map Outputs Channel 1^Data Out 9;
                              .D[10] := TIIB[IM1L0-EL6002]^COM RxPDO-Map Outputs Channel 1^Data Out 10;
                              .D[11] := TIIB[IM1L0-EL6002]^COM RxPDO-Map Outputs Channel 1^Data Out 11;
                              .D[12] := TIIB[IM1L0-EL6002]^COM RxPDO-Map Outputs Channel 1^Data Out 12;
                              .D[13] := TIIB[IM1L0-EL6002]^COM RxPDO-Map Outputs Channel 1^Data Out 13;
                              .D[14] := TIIB[IM1L0-EL6002]^COM RxPDO-Map Outputs Channel 1^Data Out 14;
                              .D[15] := TIIB[IM1L0-EL6002]^COM RxPDO-Map Outputs Channel 1^Data Out 15;
                              .D[16] := TIIB[IM1L0-EL6002]^COM RxPDO-Map Outputs Channel 1^Data Out 16;
                              .D[17] := TIIB[IM1L0-EL6002]^COM RxPDO-Map Outputs Channel 1^Data Out 17;
                              .D[18] := TIIB[IM1L0-EL6002]^COM RxPDO-Map Outputs Channel 1^Data Out 18;
                              .D[19] := TIIB[IM1L0-EL6002]^COM RxPDO-Map Outputs Channel 1^Data Out 19;
                              .D[20] := TIIB[IM1L0-EL6002]^COM RxPDO-Map Outputs Channel 1^Data Out 20;
                              .D[21] := TIIB[IM1L0-EL6002]^COM RxPDO-Map Outputs Channel 1^Data Out 21'}
    stEL6Out AT %Q*: EL6OutData22b;

    fbStateSetup: FB_StateSetupHelper;
    stDefault: ST_PositionState := (
        fVelocity := 1,
        bMoveOk := TRUE,
        bValid := TRUE
    );
END_VAR


fbStateSetup(stPositionState:=stDefault, bSetDefault:=TRUE);
fbStateSetup(stPositionState:=fbIM1L0.stOut, fPosition:=0,          sPmpsState:='IM1L0:XTES-OUT');
fbStateSetup(stPositionState:=fbIM1L0.stYag, fPosition:=-86.65,     sPmpsState:='IM1L0:XTES-YAG');
fbStateSetup(stPositionState:=fbIM1L0.stDiamond, fPosition:=-56.65, sPmpsState:='IM1L0:XTES-DIAMOND');
fbStateSetup(stPositionState:=fbIM1L0.stReticle, fPosition:=-26.65, sPmpsState:='IM1L0:XTES-RETICLE');

fbIM1L0(
    fbArbiter := GVL.fbArbiter,
    fbFFHWO := GVL.fbFastFaultOutput1,
    stYStage := Main.M20,
    stZoomStage := Main.M21,
    stFocusStage := Main.M22,
    stEl6In := stEL6In,
    stEl6Out := stEl6Out,
    sDeviceName := 'IM1L0:XTES',
    sTransitionKey := 'IM1L0:XTES-TRANSITION',
    bEnableMotion := TRUE,
    bEnableBeamParams := TRUE,
    bEnablePositionLimits := TRUE,
);

END_PROGRAM

